(* CODESYS project tc3_bacnetrev14.library
   Company: Beckhoff Automation GmbH
   DefaultNamespace: Tc3_BACnetRev14
   Version: 4.0.18.1
   Placeholder: Tc3_BACnetRev14
   Author: Beckhoff Automation GmbH
   Description: The PLC library is a collection of function blocks for programming a BACnet controller. For each BACnet object function blocks are available that are read and written via the selected properties. In general a distinction is made between function blocks for server and client objects. Function blocks for client objects have the prefix "Remote", since they enable access to remote BACnet objects on other devices. The BACnet object function blocks ascertain whether process data are valid and the BACnet controller is ready for operation.
   Title: Tc3_BACnetRev14

Project tree, tasks and I/O mapping:
  libraries: Tc2_Standard, * (Beckhoff Automation GmbH); Tc2_System, * (Beckhoff Automation GmbH); Tc2_Utilities, * (Beckhoff Automation GmbH); Tc3_BA2_Common, * (Beckhoff Automation GmbH); Tc3_Module, * (Beckhoff Automation GmbH)
  DUTs/
    Enumerations/
      [Functional]/
        data type E_BACnet_CommMode
        data type E_BACnet_CreateObjType
        data type E_BACnet_EvaluationMode
        data type E_BACnet_ServerState
      [Internal]/
        data type E_BACnet_DeviceData
        data type E_BACnet_MultistateVal
        data type E_BACnet_PlcAction
      Properties/
        Error/
          data type E_BACnet_ErrorClass
          data type E_BACnet_ErrorCode
          data type E_BACnet_ErrorType
        Event/
          data type E_BACnet_EventState
          data type E_BACnet_EventTransitionBits
          data type E_BACnet_EventType
        Recipient/
          data type E_BACnet_AddressChoice
          data type E_BACnet_RecipientChoice
        Types/
          Calendar/
            data type E_BACnet_CalendarEntryChoice
            data type E_BACnet_CalendarEntryType
          DateTime/
            data type E_BACnet_DaysOfWeekBits
            data type E_BACnet_TimeStampChoice
          LogBuffer/
            data type E_BACnet_LogRecordChoice
          Scheduler/
            data type E_BACnet_EnumerationValueChoice
            data type E_BACnet_SchedBType
            data type E_BACnet_SpecialEventChoice
            data type E_BACnet_ValueChoice
          data type E_BACnet_BinaryPV
          data type T_BACnet_MultistateValue
        data type E_BACnet_AbortReason
        data type E_BACnet_AdapterStatus
        data type E_BACnet_ClientCOVChoice
        data type E_BACnet_DataTypes
        data type E_BACnet_DeviceStatus
        data type E_BACnet_FileAccessMethod
        data type E_BACnet_LifeSafetyMode
        data type E_BACnet_LifeSafetyOperation
        data type E_BACnet_LimitEnableBits
        data type E_BACnet_LoopMode
        data type E_BACnet_NodeType
        data type E_BACnet_NotifyType
        data type E_BACnet_ObjectSupportedBits
        data type E_BACnet_PersistentDataState
        data type E_BACnet_Priority
        data type E_BACnet_ProgramError
        data type E_BACnet_ProgramRequest
        data type E_BACnet_ProgramState
        data type E_BACnet_RejectReason
        data type E_BACnet_RestartReason
        data type E_BACnet_ScaleChoice
        data type E_BACnet_Segmentation
        data type E_BACnet_ServicesSupportedBits
        data type E_BACnet_SilencedState
        data type E_BACnet_StatusFlags
        data type E_BACnet_StringEncodingTypes
      Remote/
        data type E_BACnetRM_ClientState
        data type E_BACnetRM_RequestType
      data type E_BACnet_Error
    Interfaces/
      Remote/
        Objects/
          [Base]/
            interface I_BACnetRM_Object
          [Internal]/
            interface I_BACnetRM_BaseObject: OnCOV, OnReqError, Error, ObjectID, ObjectInstance, ObjectType, ReadMode
            interface I_BACnetRM_ObjectOwner: OnBACnetRMObjectCOV, OnBACnetRMObjectStateChanged, LogMsg
        Requests/
          [Base]/
            interface I_BACnetRM_BaseReq: Send, GetRequestType, IsReady
            interface I_BACnetRM_BasicReq: SetError, SetReady
      Server/
        [Base]/
          interface I_BACnet_Object: NextSibling, PrevSibling, IsDynamic, Parent, Description, ObjectName
        [Internal]/
          interface I_BACnet_BaseObject: NextObject, Error, ObjectID, ObjectInstance, ObjectType, Ready, ReadProperty, SyncPropertyCOV, WriteProperty
          interface I_BACnet_ObjectOwner: LogMsg, SymbolName, SymbolPath, OnBACnetObjectStateChanged
        Misc/
          interface I_BACnet_Cal
          interface I_BACnet_View: AddObject, RemoveObject, FindObject
    Types/
      [ADS]/
        data type ST_BACnet_AdsConnection
      [Functional]/
        data type U_BACnet_CreateObj
      Diagnose/
        data type ST_BACnet_ConfirmedServiceDiag
        data type ST_BACnet_DiagEthStatistics
        data type ST_BACnet_Diagnosis
        data type ST_BACnet_DiagnosisTiming
        data type ST_BACnet_FrameStatistics
        data type ST_BACnet_Info
        data type ST_BACnet_ServerStatistics
        data type ST_BACnet_TcIoEthStatistic
        data type ST_BACnet_TcIoEthTxRxErrorCount
        data type ST_BACnet_UnConfirmedServiceDiag
      Properties/
        [ADS]/
          Calendar/
            data type ST_BACnet_CalendarEntry
            data type ST_BACnet_CalendarEntryDate
            data type ST_BACnet_CalendarEntryDateRange
            data type ST_BACnet_CalendarEntryWeekNDay
            data type T_BACnet_CalendarEntryTypeFilter
          DateTime/
            data type ST_BACnet_TimeStampDateTime
            data type ST_BACnet_TimeValue
            data type ST_BACnet_TimeValueBool
            data type ST_BACnet_TimeValueList
            data type ST_BACnet_TimeValueReal
          LogBuffer/
            data type ST_BACnet_LogBufferEntryReal
            data type ST_BACnet_LogBufferReal
          LogRecord/
            data type ST_BACnet_LogDatum
            data type ST_BACnet_LogDatumList
            data type ST_BACnet_LogRecord
            data type ST_BACnet_LogRecordList
          Schedule/
            data type ST_BACnet_DailySchedule
            data type ST_BACnet_ExceptionScheduleBool
            data type ST_BACnet_ExceptionScheduleCalDate
            data type ST_BACnet_ExceptionScheduleCalRef
            data type ST_BACnet_ExceptionScheduleCalWnD
            data type ST_BACnet_ExceptionScheduleEntryBool
            data type ST_BACnet_ExceptionScheduleEntryReal
            data type ST_BACnet_ExceptionScheduleReal
            data type ST_BACnet_Value
            data type ST_BACnet_ValueList
          data type ST_BACnet_CharacterStringExt
          data type ST_BACnet_CharacterStringExtListEntry
          data type ST_BACnet_LimitEnable
          data type ST_BACnet_ObjectIdentifierList
        [Raw]/
          References/
            data type ST_BACnetRaw_DeviceObjectPropertyReference
            data type ST_BACnetRaw_DeviceObjectReference
            data type ST_BACnetRaw_ObjectPropertyReference
            data type ST_BACnetRaw_SetpointReference
          ValidFields/
            data type ST_BACnetRaw_ValidFields_DeviceObjectPropertyReference
        Accumulator/
          data type ST_BACnet_Prescale
          data type ST_BACnet_Scale
          data type ST_BACnet_ScaleValue
        Calendar/
          data type T_BACnet_CalendarDateList
        Event/
          data type ST_BACnet_Event
          data type ST_BACnet_EventMessageTexts
          data type ST_BACnet_EventMessageTextStrings
          data type ST_BACnet_Events
          data type ST_BACnet_EventTimeStamps
          data type T_BACnet_EventTransitions
          data type T_BACnet_EventTransitionTexts
        EventEnrollment/
          data type ST_BACnet_EventArguments
          data type ST_BACnet_EventBinaryCoded
          data type ST_BACnet_EventOutOfRange
          data type ST_BACnet_EventParameter
          data type ST_BACnet_EventUnsignedRange
        Recipient/
          data type ST_BACnet_Address
          data type ST_BACnet_Destination
          data type ST_BACnet_Recipient
          data type ST_BACnet_RecipientEntry
          data type ST_BACnet_ValidDays
          data type T_BACnet_RecipientList
        References/
          data type ST_BACnet_ObjectPropertyReference
        Scheduler/
          data type ST_BACnet_EnumerationValueType
          data type ST_BACnet_SchedCalendar
          data type ST_BACnet_SchedException
          data type ST_BACnet_SpecialEvent
          data type ST_BACnet_SpecialEventList
          data type T_BACnet_SchedCalendar
          data type T_BACnet_SchedExceptionEntryList
          data type T_BACnet_SchedExceptionList
          data type T_BACnet_SchedWeek
        TLog/
          data type T_BACnet_TLogBuffer
        data type ST_BACnet_ClientCOV
        data type ST_BACnet_EventTransitionBits
        data type ST_BACnet_LimitEnableBits
        data type ST_BACnet_ServicesSupportedBits
        data type ST_BACnet_StatusFlagBits
        data type T_BACnet_EventTransitionPriority
        data type T_BACnet_ObjectIdentifier
        data type T_BACnet_StateText
        data type T_BACnet_StateTextArray
      Remote/
        [Internal]/
          data type ST_BACnetRM_CmdRealValue
          data type ST_BACnetRM_FifoEntry
          data type ST_BACnetRM_LastWriteValue
          data type ST_BACnetRM_PropertyValueList
          data type ST_BACnetRM_ReadEntry
          data type ST_BACnetRM_ReqPtr
          data type ST_BACnetRM_RpmListEntry
          data type ST_BACnetRM_ScanParameter
          data type ST_BACnetRM_WriteEntry
        data type ST_BACnetRM_ScanResult
  GVLs/
    global variables BACnet_Globals
    global variables BACnet_Param
  POUs/
    Dynamic Objects/
      function block FB_BACnet_DynObjectManager [ST]: EvaluateStructure, DeleteObjectEx, OnPostOnlineChange, CreateObject, CreateObjectEx, DeleteObject, Ready, Reset, CreatedObjects, FB_exit
    Helper/
      [internal]/
        Calendar/
          function F_BACnet_ToDateListEntry [ST]
        Remote/
          function F_BACnetRM_GetWriteEntrySize [ST]
          function F_BACnetRM_IsErrorSet [ST]
          function F_IsCovProperty [ST]
          function F_IsCovReadMode [ST]
          function F_IsCovReqType [ST]
        Scheduler/
          function F_BA_CalendarSchedSize [ST]
          function F_BA_ExceptionSchedSize [ST]
        String/
          function F_BACnet_ChrStrExtLen [ST]
          function F_BACnet_DecodeUCS2 [ST]
          function F_BACnet_DecodeUCS4 [ST]
          function F_BACnet_DecodeUTF8 [ST]
          function F_BACnet_EncodeUTF8 [ST]
          function F_BACnet_GetUsedStateText [ST]
          function F_BACnet_GetUsedUDINT [ST]
          function F_BACnet_UCS2ToWin1252 [ST]
          function F_BACnet_Utf8ToWin1252 [ST]
          function F_BACnet_Win1252ToUCS2 [ST]
          function F_BACnet_Win1252ToUtf8 [ST]
        Validation-Functions/
          function F_BACnet_IsAbortReasonValid [ST]
          function F_BACnet_IsErrorClassValid [ST]
          function F_BACnet_IsErrorCodeValid [ST]
          function F_BACnet_IsErrorTypeValid [ST]
          function F_BACnet_IsObjIdentifierValid [ST]
          function F_BACnet_IsPriorityValid [ST]
          function F_BACnet_IsPropIdentifierValid [ST]
          function F_BACnet_IsRejectReasonValid [ST]
          function F_BACnet_IsSchedBTypeValid [ST]
        function F_BACnet_AlignedSize [ST]
        function F_BACnet_AnalogPV [ST]
        function F_BACnet_BitFieldBit [ST]
        function F_BACnet_ChangeBitFieldBit [ST]
        function F_BACnet_ElemSize [ST]
        function F_BACnet_EndOf [ST]
        function F_BACnet_FilterErrCode [ST]
        function F_BACnet_IsBitFieldBitSet [ST]
        function F_BACnet_IsBitFieldBitSetPtr [ST]
        function F_BACnet_NextListElem [ST]
        function F_BACnet_SetBitFieldBit [ST]
        function F_BACnet_SysTimeDiff [ST]
        function F_BACnet_UnSetBitFieldBit [ST]
      Flags/
        function F_BACnet_EventEnable [ST]
        function F_BACnet_EventTransitionFlags [ST]
        function F_BACnet_GetEventTransFlagsData [ST]
        function F_BACnet_GetLimitEnFlagsData [ST]
        function F_BACnet_GetStatusFlagsData [ST]
        function F_BACnet_LimitEnable [ST]
        function F_BACnet_LimitEnableFlags [ST]
        function F_BACnet_StatusFlags [ST]
      MultiState/
        function F_BACnet_EnMultiStatePV [ST]
        function F_BACnet_MultiStatePV [ST]
      NC/
        function F_BACnet_DeviceRecipient [ST]
        function F_BACnet_EthernetRecipient [ST]
        function F_BACnet_EthernetRecipientEx [ST]
      Real/
        function F_BACnet_EnRealPV [ST]
        function F_BACnet_IsFinite [ST]
        function F_BACnet_NAN [ST]
        function F_BACnet_RealEQ [ST]
        function F_BACnet_RealGE [ST]
        function F_BACnet_RealGT [ST]
        function F_BACnet_RealLE [ST]
        function F_BACnet_RealLT [ST]
        function F_BACnet_RealNothing [ST]
        function F_BACnet_RealNull [ST]
        function F_BACnet_RealPV [ST]
        function F_BACnet_RealToStr [ST]
      References/
        function F_BACnet_Reference [ST]
        function F_BACnet_ReferenceByID [ST]
      Schedule/
        Calendar/
          function F_BACnet_SchedCalendar [ST]
        Exception/
          function F_BACnet_SchedEntry1xA [ST]
          function F_BACnet_SchedEntry1xB [ST]
          function F_BACnet_SchedEntry1xM [ST]
          function F_BACnet_SchedEntry3xA [ST]
          function F_BACnet_SchedEntry3xB [ST]
          function F_BACnet_SchedEntry3xM [ST]
          function F_BACnet_SchedEntry5xA [ST]
          function F_BACnet_SchedEntry5xB [ST]
          function F_BACnet_SchedEntry5xM [ST]
        Weekly/
          function F_BACnet_SchedWeekly1xA [ST]
          function F_BACnet_SchedWeekly1xB [ST]
          function F_BACnet_SchedWeekly1xM [ST]
          function F_BACnet_SchedWeekly3xA [ST]
          function F_BACnet_SchedWeekly3xB [ST]
          function F_BACnet_SchedWeekly3xM [ST]
          function F_BACnet_SchedWeekly5xA [ST]
          function F_BACnet_SchedWeekly5xB [ST]
          function F_BACnet_SchedWeekly5xM [ST]
      String/
        function F_BACnet_GetObjectIdString [ST]
        function block FB_BACnet_StringExtDecode [ST]
        function block FB_BACnet_StringExtEncode [ST]
      function F_BACnet_GetObjectListIndex [ST]
      function F_BACnet_GetObjId [ST]
      function F_BACnet_GetObjInstance [ST]
      function F_BACnet_GetObjType [ST]
      function block FB_BACnet_AccLimit [ST]
      function block FB_BACnet_AvgValue [ST]
      function block FB_BACnet_PidControl [ST]
      function block FB_BACnet_PT1 [ST]
    Local/
      Objects/
        [Base]/
          Basic/
            function block FB_BACnet_EventObject [ST]: OnObjectStateChanged, OnPostInit, IsReliable, AcknowledgePLC, AcknowledgeRm, AckedTransitions, EventMessageTexts, EventState, EventTimeStamps, StatusFlags, FB_init
            function block FB_BACnet_Object [ST]: OnBACnetObjectStateChanged, OnCycle, RemoveFromLinkedObjList, LogMsg, NextSibling, PrevSibling, SymbolName, SymbolPath, Close, DynamicInit, OnObjectStateChanged, OnPostInit, ValidateReference, ConcatTitle, ValidateTitles, Parent, ReadPropertyExceptionSched, ReadPropertyReference, WritePropertyExceptionSched, WritePropertyReference, Description, ObjectName, FB_init
          function block FB_BACnet_BaseAcc [ST]: OnObjectStateChanged, FB_init
          function block FB_BACnet_BaseAI [ST]: OnObjectStateChanged, FB_init
          function block FB_BACnet_BaseAO [ST]: OnObjectStateChanged, ActivePrio, FB_init
          function block FB_BACnet_BaseBI [ST]: OnObjectStateChanged, ChangeOfStateTime, TimeOfActiveTimeReset, TimeOfStateCountReset, FB_init
          function block FB_BACnet_BaseBO [ST]: OnObjectStateChanged, ActivePrio, ChangeOfStateTime, TimeOfActiveTimeReset, TimeOfStateCountReset, FB_init
          function block FB_BACnet_BaseLoop [ST]: OnObjectStateChanged, ControlledVariable, ProportionalBand, Setpoint, FB_init
          function block FB_BACnet_BaseMI [ST]: OnObjectStateChanged, StateCount, FB_init
          function block FB_BACnet_BaseMO [ST]: OnObjectStateChanged, ActivePrio, StateCount, FB_init
          function block FB_BACnet_BasePC [ST]: OnObjectStateChanged, FB_init
          function block FB_BACnet_BaseSched [ST]: OnObjectStateChanged, ReadContent, WriteContent, ObjectPropertyReferences, FB_init
          function block FB_BACnet_BaseTLog [ST]: OnObjectStateChanged, LastNotifyRecord, RecordsSinceNotification
        [Internal]/
          5P/
            function block FB_BACnet_AO_5P [ST]: OnObjectStateChanged, EnManualOperator, ValManualOperator
            function block FB_BACnet_AO_IO5P [ST]: OnObjectStateChanged, EnManualOperator, ValManualOperator
            function block FB_BACnet_AO_Raw5P [ST]: OnObjectStateChanged, EnManualOperator, ValManualOperator
            function block FB_BACnet_AV_5P [ST]: OnObjectStateChanged, EnManualOperator, ValManualOperator
            function block FB_BACnet_BO_5P [ST]: OnObjectStateChanged, EnManualOperator, ValManualOperator
            function block FB_BACnet_BO_IO5P [ST]: OnObjectStateChanged, EnManualOperator, ValManualOperator
            function block FB_BACnet_BO_Raw5P [ST]: OnObjectStateChanged, EnManualOperator, ValManualOperator
            function block FB_BACnet_BV_5P [ST]: OnObjectStateChanged, EnManualOperator, ValManualOperator
            function block FB_BACnet_MO_5P [ST]: OnObjectStateChanged, EnManualOperator, ValManualOperator
            function block FB_BACnet_MO_IO5P [ST]: OnObjectStateChanged, EnManualOperator, ValManualOperator
            function block FB_BACnet_MO_Raw5P [ST]: OnObjectStateChanged, EnManualOperator, ValManualOperator
            function block FB_BACnet_MV_5P [ST]: OnObjectStateChanged, EnManualOperator, ValManualOperator
          Property/
            Buffer/
              [Archiv]/
                function block FB_BACnet_WeeklyScheduleBuffer [ST]: ResetValue, FB_init
              Base/
                function block FB_BACnet_BaseArrayBuffer [ST]
                function block FB_BACnet_BaseListBuffer [ST]: ValidateInst
                function block FB_BACnet_BasePropertyBuffer [ST]: MemSet, MemSetBYTE, MemSetUDINT, MemSetUINT, MemSetULINT, ReadValue, ValidateInst, WriteValue, OnObjectStateChanged, ResetValue
                function block FB_BACnet_BasePropertyLogBuffer [ST]: OnObjectStateChanged
              function block FB_BACnet_DateListBuffer [ST]: FB_init
              function block FB_BACnet_EventLogBuffer [ST]: ValidateInst, FB_init
              function block FB_BACnet_ExceptionScheduleBuffer [ST]: FB_init
              function block FB_BACnet_TLMBuffer [ST]: ValidateInst, ResetValue, FB_init
              function block FB_BACnet_TrendLogBuffer [ST]: ValidateInst, ResetValue, FB_init
          function block FB_BACnet_BaseObject [ST]: OnCycle, NextObject, View_AddSubordinate, View_RemoveSubordinate, Close, Sched_ReadEntry, Sched_SetNextDay, Sched_SetNextTimeVal, Sched_WriteEntry, DeleteObject, IsInitReady, OnObjectStateChanged, OnPostOnlineChange, Acknowledge, Error, IsDynamic, ObjectID, ObjectInstance, ObjectType, Ready, State, EnableProperty, SetPropertyCount, WriteProtectProperty, AddPropertyElement, AddPropertyElementPtr, RemoveArrayElements, RemoveListElements, SetNumberOfStates, ReadProperty, ReadPropertyAckedTransitions, ReadPropertyBool, ReadPropertyByte, ReadPropertyDateList, ReadPropertyEventEnable, ReadPropertyEventParameter, ReadPropertyEventState, ReadPropertyEventTimeStamps, ReadPropertyExceptionSched, ReadPropertyLimitEnable, ReadPropertyNotifyType, ReadPropertyReal, ReadPropertyRecipientList, ReadPropertyReference, ReadPropertyStatusFlags, ReadPropertyString, ReadPropertyUDInt, ReadPropertyUnit, ReadPropertyWeeklySched, AddListElement, ApplySyncHandler, EvaluatePropSync, IncrementSyncHandlers, RequestSyncHandlers, RequestSyncHandlersEx, SyncProperty, SyncPropertyCOV, SyncPropertyIdx, SyncPropertyList, SyncPropertyPvPrio, WriteProperty, WritePropertyBool, WritePropertyByte, WritePropertyDateList, WritePropertyEventEnable, WritePropertyEventParameter, WritePropertyExceptionSched, WritePropertyLimitEnable, WritePropertyNotifyType, WritePropertyNull, WritePropertyReal, WritePropertyRealPrio, WritePropertyRecipientList, WritePropertyReference, WritePropertyReferenceList, WritePropertyReferenceList1x, WritePropertyString, WritePropertyStringIdx, WritePropertyUDInt, WritePropertyUInt, WritePropertyUnit, WritePropertyValue, WritePropertyValueEx, WritePropertyWeeklySched, FB_exit
        Experimental/
          function block FB_BACnet_ExpEventLog [ST]
          function block FB_BACnet_ExpTLM [ST]: OnObjectStateChanged, FB_init
          function block FB_BACnet_ExpTLog [ST]: Trend_LastPlcTrendEntry, Trend_NextLogDatum, Trend_NextLogRecord, OnObjectStateChanged, ReadPropertyLogBuffer, WritePropertyLogBuffer, ObjectPropertyReference, FB_init
        Primitive/
          function block FB_BACnet_INT [ST]: OnObjectStateChanged, FB_init
          function block FB_BACnet_LAV [ST]: OnObjectStateChanged, FB_init
          function block FB_BACnet_String [ST]: OnObjectStateChanged, FB_init
          function block FB_BACnet_UINT [ST]: OnObjectStateChanged, FB_init
        function block FB_BACnet_Acc [ST]: OnObjectStateChanged, FB_init
        function block FB_BACnet_Acc_IO [ST]: OnObjectStateChanged, ValueBeforeChange, ValueChangeTime
        function block FB_BACnet_Acc_Raw [ST]: OnObjectStateChanged
        function block FB_BACnet_AI [ST]: OnObjectStateChanged
        function block FB_BACnet_AI_IO [ST]: OnObjectStateChanged
        function block FB_BACnet_AI_Raw [ST]: OnObjectStateChanged
        function block FB_BACnet_AO [ST]: OnObjectStateChanged
        function block FB_BACnet_AO_IO [ST]: OnObjectStateChanged
        function block FB_BACnet_AO_Raw [ST]: OnObjectStateChanged
        function block FB_BACnet_AV [ST]: OnObjectStateChanged, ActivePrio, FB_init
        function block FB_BACnet_AV_Disp [ST]: OnObjectStateChanged, FB_init
        function block FB_BACnet_AV_Setp [ST]: OnObjectStateChanged, FB_init
        function block FB_BACnet_BI [ST]: OnObjectStateChanged
        function block FB_BACnet_BI_IO [ST]: OnObjectStateChanged
        function block FB_BACnet_BI_Raw [ST]: OnObjectStateChanged
        function block FB_BACnet_BO [ST]: OnObjectStateChanged
        function block FB_BACnet_BO_IO [ST]: OnObjectStateChanged
        function block FB_BACnet_BO_Raw [ST]: OnObjectStateChanged
        function block FB_BACnet_BV [ST]: OnObjectStateChanged, ActivePrio, ChangeOfStateTime, TimeOfActiveTimeReset, TimeOfStateCountReset, FB_init
        function block FB_BACnet_BV_Disp [ST]: OnObjectStateChanged, FB_init
        function block FB_BACnet_BV_Setp [ST]: OnObjectStateChanged, FB_init
        function block FB_BACnet_Cal [ST]: OnObjectStateChanged, ReadContent, WriteContent, FB_init
        function block FB_BACnet_Device [ST]: OnObjectStateChanged, Location, FB_init
        function block FB_BACnet_EE [ST]: OnObjectStateChanged, ReadContent, WriteContent, ObjectPropertyReference, FB_init
        function block FB_BACnet_ELog [ST]: OnObjectStateChanged, FB_init
        function block FB_BACnet_File [ST]: OnObjectStateChanged, FB_init
        function block FB_BACnet_Loop [ST]: OnObjectStateChanged, ControlledVariable, Setpoint
        function block FB_BACnet_Loop_Ref [ST]: OnObjectStateChanged, ControlledVariable, ControlledVariableReference, ManipulatedVariableReference, Setpoint, SetpointReference
        function block FB_BACnet_MI [ST]: OnObjectStateChanged
        function block FB_BACnet_MI_IO [ST]: OnObjectStateChanged
        function block FB_BACnet_MI_Raw [ST]: OnObjectStateChanged
        function block FB_BACnet_MO [ST]: OnObjectStateChanged
        function block FB_BACnet_MO_IO [ST]: OnObjectStateChanged
        function block FB_BACnet_MO_Raw [ST]: OnObjectStateChanged
        function block FB_BACnet_MV [ST]: OnObjectStateChanged, ActivePrio, StateCount, FB_init
        function block FB_BACnet_MV_Disp [ST]: OnObjectStateChanged, StateCount, FB_init
        function block FB_BACnet_MV_Setp [ST]: OnObjectStateChanged, StateCount, FB_init
        function block FB_BACnet_NC [ST]: OnObjectStateChanged, FB_init
        function block FB_BACnet_PC [ST]: OnObjectStateChanged, InputReference, FB_init
        function block FB_BACnet_PC_Raw [ST]: OnObjectStateChanged, FB_init
        function block FB_BACnet_Prog [ST]: OnObjectStateChanged, FB_init
        function block FB_BACnet_SchedA [ST]: OnObjectStateChanged, FB_init
        function block FB_BACnet_SchedB [ST]: OnObjectStateChanged, FB_init
        function block FB_BACnet_SchedM [ST]: OnObjectStateChanged, FB_init
        function block FB_BACnet_TLM [ST]: OnObjectStateChanged, ObjectPropertyReferences, FB_init
        function block FB_BACnet_TLog [ST]: OnObjectStateChanged, ObjectPropertyReference, FB_init
        function block FB_BACnet_View [ST]: AddObject, RemoveObject, Close, OnObjectStateChanged, FindObject, FB_init
      function block FB_BACnet_Server [ST]: GetObjectByID, RegisterObject, ObjectCount, ServerItf, Reset, OnPostOnlineChange, Error, Operational, Valid, ReadPropertyInt, ReadPropertyUDInt, FB_Exit
    Remote/
      Objects/
        Basic/
          [Base]/
            Basic/
              function block FB_BACnetRM_Object [ST]: OnBACnetRMObjectCOV, OnBACnetRMObjectStateChanged, LogMsg, FB_init
            function block FB_BACnetRM_BaseTLog [ST]: OnObjectStateChanged
            function block FB_BACnetRM_EventObject [ST]: OnObjectStateChanged, StatusFlags
          [Internal]/
            function block FB_BACnetRM_BaseObject [ST]: OnCOV, OnReqError, OnObjectStateChanged, Error, ObjectID, ObjectInstance, ObjectType, ReadMode, SyncProperty, SyncPropertyEnable, SyncPropertyIdx, SyncPropertyPrio, SyncPropertyPrioReal, SyncPropertyReal
          function block FB_BACnetRM_Acc [ST]: OnObjectStateChanged, FB_init
          function block FB_BACnetRM_AI [ST]: OnObjectStateChanged, FB_init
          function block FB_BACnetRM_AO [ST]: OnObjectStateChanged, FB_init
          function block FB_BACnetRM_AV [ST]: OnObjectStateChanged, FB_init
          function block FB_BACnetRM_AV_Disp [ST]: OnObjectStateChanged, FB_init
          function block FB_BACnetRM_AV_Setp [ST]: OnCOV, OnObjectStateChanged, FB_init
          function block FB_BACnetRM_Avg [ST]: OnObjectStateChanged, FB_init
          function block FB_BACnetRM_BI [ST]: OnObjectStateChanged, FB_init
          function block FB_BACnetRM_BO [ST]: OnObjectStateChanged, FB_init
          function block FB_BACnetRM_BV [ST]: OnObjectStateChanged, FB_init
          function block FB_BACnetRM_BV_Disp [ST]: OnObjectStateChanged, FB_init
          function block FB_BACnetRM_BV_Setp [ST]: OnCOV, OnObjectStateChanged, FB_init
          function block FB_BACnetRM_Cal [ST]: OnObjectStateChanged, FB_init
          function block FB_BACnetRM_Cmd [ST]: OnObjectStateChanged, FB_init
          function block FB_BACnetRM_Device [ST]: OnObjectStateChanged, FB_init
          function block FB_BACnetRM_EE [ST]: OnObjectStateChanged, FB_init
          function block FB_BACnetRM_ELog [ST]: FB_init
          function block FB_BACnetRM_File [ST]: OnObjectStateChanged, FB_init
          function block FB_BACnetRM_Group [ST]: OnObjectStateChanged, FB_init
          function block FB_BACnetRM_Loop [ST]: OnObjectStateChanged, FB_init
          function block FB_BACnetRM_MI [ST]: OnObjectStateChanged, FB_init
          function block FB_BACnetRM_MO [ST]: OnObjectStateChanged, FB_init
          function block FB_BACnetRM_MV [ST]: OnObjectStateChanged, FB_init
          function block FB_BACnetRM_MV_Disp [ST]: OnObjectStateChanged, FB_init
          function block FB_BACnetRM_MV_Setp [ST]: OnCOV, OnObjectStateChanged, FB_init
          function block FB_BACnetRM_NC [ST]: FB_init
          function block FB_BACnetRM_PC [ST]: OnObjectStateChanged, FB_init
          function block FB_BACnetRM_Prog [ST]: OnObjectStateChanged, FB_init
          function block FB_BACnetRM_SchedA [ST]: OnObjectStateChanged, FB_init
          function block FB_BACnetRM_SchedB [ST]: OnObjectStateChanged, FB_init
          function block FB_BACnetRM_SchedM [ST]: OnObjectStateChanged, FB_init
          function block FB_BACnetRM_TLM [ST]: OnObjectStateChanged, FB_init
          function block FB_BACnetRM_TLog [ST]: OnObjectStateChanged, FB_init
        Convenience/
          function block FB_BACnetRM_CnvLoop [ST]: OnObjectStateChanged
        Experimental/
          function block FB_BACnetRM_ExpAV01 [ST]: OnObjectStateChanged
          function block FB_BACnetRM_ExpAV02 [ST]
        Primitive/
          function block FB_BACnetRM_BitString [ST]: OnObjectStateChanged, FB_init
          function block FB_BACnetRM_ByteArr [ST]: OnObjectStateChanged, FB_init
          function block FB_BACnetRM_Date [ST]: OnObjectStateChanged, FB_init
          function block FB_BACnetRM_DateP [ST]: OnObjectStateChanged, FB_init
          function block FB_BACnetRM_DateTime [ST]: OnObjectStateChanged, FB_init
          function block FB_BACnetRM_DateTimeP [ST]: OnObjectStateChanged, FB_init
          function block FB_BACnetRM_Int [ST]: OnObjectStateChanged, FB_init
          function block FB_BACnetRM_LAV [ST]: OnObjectStateChanged, FB_init
          function block FB_BACnetRM_String [ST]: OnObjectStateChanged, FB_init
          function block FB_BACnetRM_Time [ST]: OnObjectStateChanged, FB_init
          function block FB_BACnetRM_TimeP [ST]: OnObjectStateChanged, FB_init
          function block FB_BACnetRM_UInt [ST]: OnObjectStateChanged, FB_init
      Properties/
        [Base]/
          function block FB_BACnetRM_BaseProperty [ST]: SetBusy, SetError, SetReady, OnExecuteChange, Free, Busy, Error, Ready, Request, Valid
        function block FB_BACnetRM_ReadProperty [ST]: OnExecuteChange, Free, Valid, FB_exit
        function block FB_BACnetRM_ReadPropertyEx [ST]
        function block FB_BACnetRM_WriteProperty [ST]: OnExecuteChange, Free, Valid, FB_exit
        function block FB_BACnetRM_WritePropertyEx [ST]
      Requests/
        [Internal]/
          [Base]/
            function block FB_BACnetRM_ReqBase [ST]: OnError, Valid, GetRequestType, IsReady, Send
            function block FB_BACnetRM_ReqBasic [ST]: OnSendPropertyDataRequest, InitTimer, SetBusy, SetError, SetReady, TcAddRef, TcQueryInterface, TcRelease, CopyRemoteData, ProcessResult, Send, StartTimer, GetRequestType, IsReady
          function block FB_BACnetRM_ReqAckAlarm [ST]: OnSendPropertyDataRequest, Send, TcAddRef, TcQueryInterface, TcRelease, UpdateTimeStamp, GetRequestType, IsReady
          function block FB_BACnetRM_ReqCov [ST]: AddCovSlave, Send, ProcessResult, StartTimer, GetRequestType, IsReady, FB_Exit, Master, SendSubscription
          function block FB_BACnetRM_ReqFifo [ST]: AddFifoReq, ProcessReadFifo, ProcessWriteFifo, Valid, FB_Exit
          function block FB_BACnetRM_ReqListAdd [ST]: Send, ProcessResult, GetRequestType, IsReady
          function block FB_BACnetRM_ReqListRem [ST]: Send, ProcessResult, GetRequestType
          function block FB_BACnetRM_ReqRead [ST]: Send, OnError, ProcessResult, GetRequestType
          function block FB_BACnetRM_ReqRpm [ST]: Send, UpdateRequest, Free, OnError, ProcessResult, GetRequestType, _WritePropEntry, FB_exit
          function block FB_BACnetRM_ReqWpm [ST]: Send, UpdateRequest, Free, OnError, ProcessResult, GetRequestType, FB_exit
          function block FB_BACnetRM_ReqWrite [ST]: Send, OnError, ProcessResult, GetRequestType, IsReady
      function block FB_BACnet_Client [ST]: OnCOV, OnReqError, OnRequestComplete, AddReadEntry, AddWriteEntry, AddFifoReadReq, AddFifoWriteReq, UpdateRequests, CreateReadReq, CreateReqList, DeleteReqList, OptimizeCOV, OnPostOnlineChange, Error, ObjectID, ObjectInstance, ObjectType, OpenRequestCount, ReadMode, Ready, State, FB_Exit
    function block FB_BACnet_Adapter [ST]: GetDiagnosis, ResetDiagnosis, Device, Error, GetScanResult, StartScan, StartScanEx, TimeSync, FB_exit, FB_init
  TEST/
    TestPackage/
      Samples/
        Objects/
          Local/
            function block FB_BACnet_SmplAV01 [ST]: OnObjectStateChanged
            function block FB_BACnet_SmplBO01 [ST]
          Remote/
            function block FB_BACnetRM_SmplAV01 [ST]: OnObjectStateChanged
        Project Structure/
          PRG02/
            TEMPLATES/
              Custom/
                H/
                  HtgCirABC123/
                    function block FB_BA_HtgCirABC123 [CFC]: FB_init
                    function block FB_BA_HtgCirABC123_Vlv [CFC]: FB_init
                  HtgCirTZU555/
                    function block FB_BA_HtgCirTZU555 [CFC]: FB_init
                    function block FB_BA_HtgCirTZU555_Pu [CFC]: FB_init
              Standard/
                AC/
                  function block FB_BACnet_AC01 [CFC]: FB_init
                H/
                  function block FB_BACnet_HtgCir01 [CFC]: FB_init
                Universal/
                  Valve/
                    function block FB_Bnet_Vlv_014 [CFC]: FB_init
            program MAIN_PRG02 [ST]
      Templates/
        HeatSupply/
          HeatingCircuit/
            Plants/
              function block FB_Bnet_H_HtgCir_01 [CFC]: FB_init
            function block FB_Bnet_H_HtgCir_HtgLmt [CFC]: FB_init
            function block FB_Bnet_H_HtgCir_Sp [CFC]: FB_init
            function block FB_MMUX_R04 [ST]
            function block FB_Swi2P [ST]
          data type E_xEnergyLvl
          data type E_xEnergyLvlA
          function block FB_Bnet_H_OpM [CFC]: FB_init
          function block FB_PrioSwi_B04 [ST]
          function block FB_PrioSwi_UDI08 [ST]
        Internal/
          function block FB_BACnet_Server_NC01 [ST]
        Universal/
          AntiBlocking/
            function F_RemSecsTon [ST]
            function block FB_AntBlkg [ST]
            function block FB_Bnet_AntiBlocking [CFC]: FB_init
          Control/
            DelayOff/
              function block FB_Bnet_DlyOff [CFC]: FB_init
            Scale/
              function block FB_Bnet_Scale_04 [CFC]: FB_init
              function block FB_Chrct04 [ST]
          Pump/
            1st/
              function block FB_Bnet_Pu1st [CFC]: FB_init
          Valve/
            function block FB_Bnet_Vlv_013 [CFC]: FB_init
        global variables Const
      TestFBs/
        RT/
          function block FB_ArrayHtgCir [ST]: FB_init
          function block FB_ArrayTest [ST]: FB_init
        function block FB_ClientTest [ST]
      program _MAIN [ST]
      program BACKUP [ST]
      program CLIENT [ST]
      program DYN_OBJECTS [ST]
      program PERFORMANCE [ST]
      program PERFORMANCE_MIX [ST]
      program PLANT_DEMO [ST]: FB_init
      program RT [ST]
    program CLIENT_Andreas [ST]
    program CLIENT_Marco [ST]
    program Experimental [ST]
    program MAIN [ST]
    program TEMP [ST]
  Version/
    global variables Global_Version
*)

// DUTs/Enumerations/[Functional]/E_BACnet_CommMode
{attribute 'qualified_only'}
TYPE E_BACnet_CommMode :
(
	eAuto	:= 0,
	
	eCov	:= 1,
	eCovC	:= 2,
	eCovU	:= 3,
	eRp		:= 4,
	eRpm	:= 5
);
END_TYPE

// DUTs/Enumerations/[Functional]/E_BACnet_CreateObjType
{attribute 'qualified_only'}
TYPE E_BACnet_CreateObjType:
(
	eAnalogInputRaw,
	eAnalogOutputRaw,
	eAnalogOutputRaw5P,
	eAnalogValue,
	eAnalogValue5P,
	eAnalogValueDisp,
	eAnalogValueSetp,
	
	eBinaryInputRaw,
	eBinaryOutputRaw,
	eBinaryOutputRaw5P,
	eBinaryValue,
	eBinaryValue5P,
	eBinaryValueDisp,
	eBinaryValueSetp,
	
	eMultiStateInputRaw,
	eMultiStateOutputRaw,
	eMultiStateOutputRaw5P,
	eMultiStateValue,
	eMultiStateValue5P,
	eMultiStateValueDisp,
	eMultiStateValueSetp,
	
	eCalendar,
	eDevice,
	eFile,
	eLoop,
	eNotificationClass,
	eProg,
	eScheduleAnalog,
	eScheduleBinary,
	eScheduleMultistate,
	eAccumulator,
	ePulseConverter,
	eStructuredView
);
END_TYPE

// DUTs/Enumerations/[Functional]/E_BACnet_EvaluationMode
{attribute 'hide'}
{attribute 'qualified_only'}
TYPE E_BACnet_EvaluationMode :
(
	// [Management] Dynamic Objects:
	eDeleteObjects			:= 0,
	eCycle					:= 1
);
END_TYPE

// DUTs/Enumerations/[Functional]/E_BACnet_ServerState
{attribute 'qualified_only'}
TYPE E_BACnet_ServerState :
(
	Invalid					:= 0,
	
	eInitServer				:= 1,
	eInitDefObjs			:= 2,
	eInitUndefObjs			:= 3,
	eInitDefRefObjs			:= 4,
	eInitUndefRefObjs		:= 5,
	eOperation				:= 6
	
) BYTE;
END_TYPE

// DUTs/Enumerations/[Internal]/E_BACnet_DeviceData
{attribute 'hide'}
{attribute 'qualified_only'}
TYPE E_BACnet_DeviceData :
(
	eGetDiagnosis	:= 16#00000001,
	eResetDiagnosis	:= 16#80000001,
	eGetScanResult	:= 16#00000002,
	eGetIPSettings	:= 16#00000003,
	eSetIPSettings	:= 16#80000003,
	eGetBDT			:= 16#00000004,
	eSetBDT			:= 16#80000004,
	eGetFDT			:= 16#00000005,
	eSetPlcOID		:= 16#80000006,
	eSetPlcAdsPort	:= 16#80000007
	
) UDINT;
END_TYPE

// DUTs/Enumerations/[Internal]/E_BACnet_MultistateVal
{attribute 'hide'}
{attribute 'qualified_only'}
TYPE E_BACnet_MultistateVal:
(
	eNull					:= 16#0,
	eMin					:= 1,
	eNothing				:= 16#FFFFFFFF
) UDINT;
END_TYPE

// DUTs/Enumerations/[Internal]/E_BACnet_PlcAction
{attribute 'hide'}
{attribute 'qualified_only'}
TYPE E_BACnet_PlcAction :
(
	eIdle,
	eStart,
	eSuspend,
	eCreateFinish
) UINT;
END_TYPE

// DUTs/Enumerations/Properties/Error/E_BACnet_ErrorClass
{attribute 'qualified_only'}
{warning disable C0125}
TYPE E_BACnet_ErrorClass :
(
	eDevice					:= 0,
	eObject					:= 1,
	eProperty				:= 2,
	eResources				:= 3,
	eSecurity				:= 4,
	eServices				:= 5,
	eVt						:= 6,
	eCommunication			:= 7,
	
	eErrorClassUnknown	    := 255,
	
	NoError					:= 256,
	First					:= eDevice,
	Last					:= eCommunication,
	Count					:= (Last - First + 1)
);
END_TYPE
{warning restore C0125}

// DUTs/Enumerations/Properties/Error/E_BACnet_ErrorCode
{attribute 'qualifiedOnly'}
{warning disable C0125}
TYPE E_BACnet_ErrorCode :
(
	eOther										:= 0,
	eAuthenticationFailed						:= 1,
	eConfigurationInProgress					:= 2,
	eDeviceBusy									:= 3,
	eDynamicCreationNotSupported				:= 4,
	eFileAccessDenied							:= 5,
	eIncompatibleSecurityLevels					:= 6,
	eInconsistentParameters						:= 7,
	eInconsistentSelectionCriterion				:= 8,
	eInvalidDataType							:= 9,
	eInvalidFileAccessMethod					:= 10,
	eInvalidFileStartPosition					:= 11,
	eInvalidOperatorName						:= 12,
	eInvalidParameterDataType					:= 13,
	eInvalidTimeStamp							:= 14,
	eKeyGenerationError							:= 15,
	eMissingRequiredParameter					:= 16,
	eNoObjectsOfSpecifiedType					:= 17,
	eNoSpaceForObject							:= 18,
	eNoSpaceToAddListElement					:= 19,
	eNoSpaceToWriteProperty						:= 20,
	eNoVTSessionsAvailable						:= 21,
	ePropertyIsNotAList							:= 22,
	eObjectDeletionNotPermitted					:= 23,
	eObjectIdentifierAlreadyExists				:= 24,
	eOperationalProblem							:= 25,
	ePasswordFailure							:= 26,
	eReadAccessDenied							:= 27,
	eSecurityNotSupported						:= 28,
	eServiceRequestDenied						:= 29,
	eTimeout									:= 30,
	eUnknownObject								:= 31,
	eUnknownProperty							:= 32,
	eUnknownVTClass								:= 34,
	eUnknownVTSession							:= 35,
	eUnsupportedObjectType						:= 36,
	eValueOutOfRange							:= 37,
	eVtSessionAlreadyClosed						:= 38,
	eVtSessionTerminationFailure				:= 39,
	eWriteAccessDenied							:= 40,
	eCharacterSetNotSupported					:= 41,
	eInvalidArrayIndex							:= 42,
	eCovSubscriptionFailed						:= 43,
	eNotCovProperty								:= 44,
	eOptionalFunctionalityNotSupported			:= 45,
	eInvalidConfigurationData					:= 46,
	eDatatypeNotSupported						:= 47,
	eDuplicateName								:= 48,
	eDuplicateObjectId							:= 49,
	ePropertyIsNotAnArray						:= 50,
	eAbortBufferOverflow						:= 51,
	eAbortInvalidAPDUInThisState				:= 52,
	eAbortPreemptedByHigherPriorityTask			:= 53,
	eAbortSegmentationNotSupported				:= 54,
	eAbortProprietary							:= 55,
	eAbortOther									:= 56,
	eInvalidTag									:= 57,
	eNetworkDown								:= 58,
	eRejectBufferOverflow						:= 59,
	eRejectInconsistentParameters				:= 60,
	eRejectInvalidParameterDataType				:= 61,
	eRejectInvalidTag							:= 62,
	eRejectMissingRequiredParameter				:= 63,
	eRejectParameterOutOfRange					:= 64,
	eRejectTooManyArguments						:= 65,
	eRejectUndefinedEnumeration					:= 66,
	eRejectUnrecognizedService					:= 67,
	eRejectProprietary							:= 68,
	eRejectOther								:= 69,
	eUnknownDevice								:= 70,
	eUnknownRoute								:= 71,
	eValueNotInitialized						:= 72,
	eInvalidEventState							:= 73,
	eNoAlarmConfigured							:= 74,
	eLogBufferFull								:= 75,
	eLoggedValuePurged							:= 76,
	eNoPropertySpecified						:= 77,
	eNotConfiguredForTriggeredLogging			:= 78,
	eUnknownSubscription						:= 79,
	eParameterOutOfRange						:= 80,
	eListElementNotFound						:= 81,
	eBusy										:= 82,
	eCommunicationDisabled						:= 83,
	eUnknownFileSize							:= 122,
	eAbortAPDUTooLong							:= 123,
	eAbortApplicationExceededReplyTime			:= 124,
	eAbortOutOfResources						:= 125,
	eAbortTsmTimeout							:= 126,
	eAbortWindowSizeOutOfRange					:= 127,
	eFileFull									:= 128,
	eInconsistentConfiguration					:= 129,
	eInconsistentObjectType						:= 130,
	eInternalError								:= 131,
	eNotConfigured								:= 132,
	eOutOfMemory 								:= 133,
	
	NoError										:= 256,
	First										:= eOther,
	Last										:= eOutOfMemory,
	Count										:= (Last - First + 1)
);
END_TYPE
{warning restore C0125}

// DUTs/Enumerations/Properties/Error/E_BACnet_ErrorType
{attribute 'qualified_only'}
{warning disable C0125}
TYPE E_BACnet_ErrorType :
(
	eError,
	eReject,
	eAbort,
	
	First					:= eError,
	Last					:= eAbort,
	Count					:= (Last - First + 1)
);
END_TYPE
{warning restore C0125}

// DUTs/Enumerations/Properties/Event/E_BACnet_EventState
{attribute 'qualified_only'}
TYPE E_BACnet_EventState:
(
	eNormal := 0,
	eFault := 1,
	eOffnormal := 2,
	eHighLimit := 3,
	eLowLimit := 4,
	eLifeSafetyAlarm := 5
) UDINT;
END_TYPE

// DUTs/Enumerations/Properties/Event/E_BACnet_EventTransitionBits
{attribute 'qualified_only'}
TYPE E_BACnet_EventTransitionBits:
(
	Invalid			:= -1,
	
	eToOffnormal	:= 0,
	eToFault		:= 1,
	eToNormal		:= 2
);
END_TYPE

// DUTs/Enumerations/Properties/Event/E_BACnet_EventType
{attribute 'qualified_only'}
TYPE E_BACnet_EventType:
(
	Invalid := -1,
	
	eChangeOfBitstring := 0,
	eChangeOfState := 1,
	eChangeOfValue := 2,
	eCommandFailure := 3,
	eFloatingLimit := 4,
	eOutOfRange := 5,
	eComplexEventType := 6,
	eDeprecated7 := 7,
	eChangeOfLifeSafety := 8,
	eEnumeration := 9,
	eBufferReady := 10,
	eUnsignedRange := 11,
	eReserved12 := 12,
	eAccessEvent := 13,
	eDoubleOutOfRange := 14,
	eSignedOutOfRange := 15,
	eUnsignedOutOfRange := 16,
	eChangeOfCharacterstring := 17,
	eChangeOfStateFlags := 18,
	eChangeOfReliability := 19
);
END_TYPE

// DUTs/Enumerations/Properties/Recipient/E_BACnet_AddressChoice
{attribute 'qualified_only'}
TYPE E_BACnet_AddressChoice :
(
	eEthernet:=0,
	eArcnet:=1,
	eMsTp:=2,
	eLonTalk:=3,
	eLonTalkNeuronId:=4,
	eAddress_3:=5,
	eAddress_4:=6,
	eAddress_5:=7,
	eBroadcast:=8
);
END_TYPE

// DUTs/Enumerations/Properties/Recipient/E_BACnet_RecipientChoice
{attribute 'qualified_only'}
TYPE E_BACnet_RecipientChoice :
(
	eDevice,
	eAddress
);
END_TYPE

// DUTs/Enumerations/Properties/Types/Calendar/E_BACnet_CalendarEntryChoice
{attribute 'qualified_only'}
TYPE E_BACnet_CalendarEntryChoice :
(
(*
	BACnetDate              DATE;
	BACnetDateRange   		dateRange;
	BACnetWeekNDay          weekNDay;
*)
	eDate,
	eDateRange,
	eWeekNDay
);
END_TYPE

// DUTs/Enumerations/Properties/Types/Calendar/E_BACnet_CalendarEntryType
{attribute 'qualified_only'}
TYPE E_BACnet_CalendarEntryType : (* Not a BACnet-Stack type! *)
(
	eNone,
	eRef,
	eDate,
	eDateRange,
	eWeekNDay
);
END_TYPE

// DUTs/Enumerations/Properties/Types/DateTime/E_BACnet_DaysOfWeekBits
{attribute 'qualified_only'}
TYPE E_BACnet_DaysOfWeekBits :
(
	Invalid		:= -1,
	
	eBitMonday		:= 0,
	eBitTuesday		:= 1,
	eBitWednesday	:= 2,
	eBitThursday	:= 3,
	eBitFriday		:= 4,
	eBitSaturday	:= 5,
	eBitSunday		:= 6
);
END_TYPE

// DUTs/Enumerations/Properties/Types/DateTime/E_BACnet_TimeStampChoice
{attribute 'qualified_only'}
TYPE E_BACnet_TimeStampChoice :
(
	eTsTime,
    eSequenceNumber,
    eDateTime
);
END_TYPE

// DUTs/Enumerations/Properties/Types/LogBuffer/E_BACnet_LogRecordChoice
{attribute 'qualified_only'}
TYPE E_BACnet_LogRecordChoice :
(
(*
enum BACnetLogRecordChoice
{
      logStatus,              // [0] BACnetLogStatus,
      booleanValue,           // [1] BOOL,
      realValue,              // [2] REAL,
      enumValue,              // [3] ENUMERATED, __ Optionally limited to 32 bits
      unsignedValue,          // [4] Unsigned, __ Optionally limited to 32 bits
      signedValue,            // [5] INTEGER, __ Optionally limited to 32 bits
      bitstringValue,         // [6] BIT STRING, __ Optionally limited to 32 bits
      nullValue,              // [7] NULL,
      failure,                // [8] Error,
      timeChange,             // [9] REAL,
      anyValue,               // [10] ABSTRACT_SYNTAX.&Type __ Optional
};
*)
	eLogStatus 	:= 0, (* BACnetLogStatus *)
	eBooleanValue := 1, (*  BOOL, *)
	eRealValue	:= 2, (*  REAL, *)
	eEnumValue	:= 3, (*  ENUMERATED, __ Optionally limited TO 32 bits *)
	eUnsignedValue:= 4, (*  Unsigned, __ Optionally limited TO 32 bits *)
	eSignedValue	:= 5, (*  INTEGER, __ Optionally limited TO 32 bits *)
	eBitstringValue:= 6, (*  BIT STRING, __ Optionally limited TO 32 bits *)
	eNullValue	:= 7, (*  NULL, *)
	eFailure		:= 8, (*  Error, *)
	eTimeChange	:= 9, (*  REAL, *)
	eAnyValue		:= 10 (*  ABSTRACT_SYNTAX.&TYPE __ Optional *)
);
END_TYPE

// DUTs/Enumerations/Properties/Types/Scheduler/E_BACnet_EnumerationValueChoice
{attribute 'qualified_only'}
TYPE E_BACnet_EnumerationValueChoice :
(
	  eEnum := 0,
      eBinaryPV := 1,
      eEngineeringUnits := 2
)UDINT;
END_TYPE

// DUTs/Enumerations/Properties/Types/Scheduler/E_BACnet_SchedBType
{attribute 'qualified_only'}
{warning disable C0125}
TYPE E_BACnet_SchedBType :
(
	Invalid				:= 0,
	
	eBinaryPV			:= 1,
	eBool				:= 2,
	
	First				:= eBinaryPV,
	Last				:= eBool,
	Count				:= (Last - First + 1)
);
END_TYPE
{warning restore C0125}

// DUTs/Enumerations/Properties/Types/Scheduler/E_BACnet_SpecialEventChoice
{attribute 'qualified_only'}
TYPE E_BACnet_SpecialEventChoice :
(
	eCalendarEntry,
	eCalendarReference
);
END_TYPE

// DUTs/Enumerations/Properties/Types/Scheduler/E_BACnet_ValueChoice
{attribute 'qualified_only'}
{warning disable C0125}
TYPE E_BACnet_ValueChoice :
(
	Invalid						:= -1,
	
	eNullValue					:= 0,
	eBoolValue					:= 1,
	eUnsignedValue				:= 2,
	eSignedValue				:= 3,
	eRealValue					:= 4,
	eDoubleValue				:= 5,
	eOctedStringValue			:= 6,
	eCharStringValue			:= 7,
	eObjectIdentifierValue 		:= 8,		// but DataType is 0x0C
	eEnumerationValue			:= 9,
	eMaxBACnetValueChoice		:= 10
	
	//XFirst						:= eNullValue,
	//XLast						:= eMaxBACnetValueChoice,
	//Count						:= (Last - First + 1)
);
END_TYPE
{warning restore C0125}

// DUTs/Enumerations/Properties/Types/E_BACnet_BinaryPV
{attribute 'qualified_only'}
TYPE E_BACnet_BinaryPV:
(
	eInactive := 0,
	eActive := 1,
	eNull := 2,
	eNothing := 16#FFFF
);
END_TYPE

// DUTs/Enumerations/Properties/Types/T_BACnet_MultistateValue
TYPE T_BACnet_MultistateValue : ARRAY[1..BACnet_Param.nMultistate_StateCount] OF UDINT; END_TYPE

// DUTs/Enumerations/Properties/E_BACnet_AbortReason
{attribute 'qualified_only'}
{warning disable C0125}
TYPE E_BACnet_AbortReason :
(
	Invalid								:= -1,
	NoReason							:= 256,
	
	eOther								:= 0,
	eBufferOverflow						:= 1,
	eInvalidAPDUInThisState				:= 2,
	ePreemptedByHigherPriorityTask		:= 3,
	eSegmentationNotSupported			:= 4,
	eWindowSizeOutOfRange				:= 7,
	eApplicationExceededReplyTime		:= 8,
	eOutOfResources						:= 9,
	eTSMTimeout							:= 10,
	eAPDUTooLong						:= 11,
	
	First								:= eOther,
	Last								:= eAPDUTooLong,
	Count								:= (Last - First + 1)
);
END_TYPE
{warning restore C0125}

// DUTs/Enumerations/Properties/E_BACnet_AdapterStatus
{attribute 'qualified_only'}
TYPE E_BACnet_AdapterStatus :
(
	eInit				:= 16#0,
	eCheckIpAddr		:= 16#1,
	eCheckParam			:= 16#2,
	eGetGatewayMAC		:= 16#3,
	eWaitGatewayMAC		:= 16#4,
	eComplete			:= 16#8
);
END_TYPE

// DUTs/Enumerations/Properties/E_BACnet_ClientCOVChoice
{attribute 'qualified_only'}
{attribute 'strict'}
TYPE E_BACnet_ClientCOVChoice :
(
	eCovNull := 0,
	eCovReal := 1
);
END_TYPE

// DUTs/Enumerations/Properties/E_BACnet_DataTypes
{attribute 'qualified_only'}
TYPE E_BACnet_DataTypes:
(
	Invalid := -1,
	
	eNull := 0,
	eBool := 1,
	eUnsignedInteger := 2,
	eSignedInteger := 3,
	eReal := 4,
	eDouble := 5,
	eOctetString := 6,
	eCharacterStringExt := 7,
	eBitString := 8,
	eEnumerated := 9,
	eDate := 10,
	eTime := 11,
	eObjectIdentifier := 12,
	eDateTime := 14,
	eArrayIndex := 15,
	eCalendarEntry := 16,
	eObjectType := 17,
	eEventTransitionBits := 18,
	eActionList := 19,
	eStatusFlags := 20,
	eEventState := 21,
	eReliability := 22,
	ePolarity := 23,
	eEngineeringUnits := 25,
	ePriorityValue := 26,
	eLimitEnable := 27,
	eNotifyType := 29,
	eTimeStamp := 30,
	eDeviceObjectPropertyReference := 31,
	eDeviceStatus := 32,
	eServicesSupported := 33,
	eObjectTypesSupported := 34,
	eSegmentation := 35,
	eVTClass := 36,
	eVTSession := 37,
	eSessionKey := 38,
	eRecipient := 39,
	eAddressBinding := 40,
	eCOVSubscription := 41,
	eEventType := 42,
	eEventParameter := 43,
	eFileAccessMethod := 44,
	eReadAccessSpecification := 45,
	eReadAccessResult := 46,
	eObjectPropertyReference := 47,
	eSetpointReference := 48,
	eDestination := 49,
	eProgramState := 50,
	eProgramRequest := 51,
	eProgramError := 52,
	eDateRange := 53,
	eDailySchedule := 54,
	eSpecialEvent := 55,
	eClientCOV := 56,
	eLogRecord := 57,
	eLifeSafetyState := 58,
	eLifeSafetyMode := 59,
	eSilencedState := 60,
	eLifeSafetyOperation := 61,
	eBinaryPV := 62,
	eDaysOfWeek := 63,
	eWeekNDay := 64,
	eTimeValue := 65,
	eValue := 66,
	eAddress := 67,
	ePropertyIdentifier := 68,
	eEnumerationValueType := 69,
	eBitFieldBit := 70,
	eLogDatum := 71,
	eAnyType := 72,
	ePresentValue := 73,
	eContextTag := 74,
	eValueChoice := 75,
	eLogStatus := 76,
	eRecipientProcess := 77,
	eSubscribeCOVPropertyRequest := 78,
	ePropertyReference := 79,
	ePropertyResult := 80,
	eDeviceObjectPropertyValue := 81,
	eCOVNotificationRequest := 82,
	eEventNotificationRequest := 83,
	eNotificationParameters := 84,
	eChangeOfBitstring := 85,
	eChangeOfState := 86,
	eChangeOfValue := 87,
	eCommandFailure := 88,
	eFloatingLimit := 89,
	eOutOfRange := 90,
	ePropertyValue := 91,
	eComplexTag := 92,
	eChangeOfLifeSafety := 93,
	eExtended := 94,
	eBufferReady := 95,
	eUnsignedRange := 96,
	ePropertyResultValue := 97,
	eServiceCOVPropSubscription := 98,
	eServiceCOVSubscription := 99,
	eCOVNotification := 100,
	eAcknowledgeAlarmRequest := 101,
	eVTOpenRequest := 102,
	ePrescale := 103,
	eScale := 104,
	eAction := 105,
	eError := 106,
	eErrorType := 107,
	eErrorClass := 108,
	eErrorCode := 109,
	eRejectReason := 110,
	eAbortReason := 111,
	eBDTEntry := 112,
	eIpEntry := 113,
	eMaskEntry := 114,
	eEthernetAddress := 115,
	eLonTalkAddress := 116,
	eLonTalkNeuronId := 117,
	eNodeType := 118,
	eDeviceObjectReference := 119,
	eActionCommand := 120,
	eGetEventInformation := 121,
	eGetEnrollmentSummaryCriteria := 122,
	eGetEnrollmentSummaryCriteriaResponse := 123,
	eDeviceCommunicationControl := 124,
	eInt16 := 125,
	eUInt16 := 126,
	eUInt8 := 127,
	eTypeInt8 := 128,
	eByte := 129,
	eFDTEntry := 130,
	eAddress_3 := 131,
	eAddress_4 := 132,
	eAddress_5 := 133,
	ePersistentDataState := 134,
	eFallbackRealValue := 135,
	eFallbackBinaryValue := 136,
	eRealNull := 137,						// PresentValue in AnalogObj
	eEnumeratedNull := 138,					// PresentValue in BinaryObj
	eUnsignedIntegerNull := 139,			// PresentValue in Multistate
	eUnknown := 140,
	eDiagnosisPerformance := 200,
	eDiagnosisEthStatistics := 201,
	eFrameStatistics := 202,
	eInfo := 203,
	eDiagnosis := 204,
	eTcIoEthStatistic := 205,
	eTcIoEthTxRxErrorCount := 206,
	eTcIoEthPortStatistic := 207,
	eServerStatistics := 208,
	eFrameServicesDiag := 209,
	eUnsignedIntegerArr := 258,
	eCharacterStringExtArr := 263,
	eObjectIdentifierArr := 268,
	eCalendarEntryArr := 272,
	eActionListArr := 275,
	ePriorityValueArr := 282,
	eTimeStampArr := 286,
	eDeviceObjectPropertyReferenceArr := 287,
	eVTClassArr := 292,
	eVTSessionArr := 293,
	eSessionKeyArr := 294,
	eRecipientArr := 295,
	eAddressBindingArr := 296,
	eCOVSubscriptionArr := 297,
	eReadAccessSpecificationArr := 301,
	eReadAccessResultArr := 302,
	eDestinationArr := 305,
	eSpecialEventArr := 311,
	eLogRecordArr := 313,
	eLifeSafetyStateArr := 314,
	eTimeValueArr := 321,
	eUnsignedIntegerList := 514,
	eCharacterStringExtList := 519,
	eReadAccessSpecificationList := 557,
	eReadAccessResultList := 558,
	eSpecialEventList := 567,
	eLogRecordList := 569,
	eTimeValueList := 577,
	eValueList := 578,
	eLogDatumList := 583,
	ePropertyReferenceList := 591,
	ePropertyResultList := 592,
	eCOVNotificationRequestList := 594,
	eEventNotificationRequestList := 595,
	ePropertyValueList := 603,
	eDailyScheduleList := 1089
);
END_TYPE

// DUTs/Enumerations/Properties/E_BACnet_DeviceStatus
{attribute 'qualified_only'}
TYPE E_BACnet_DeviceStatus:
(
	Invalid					:= -1,
	
	eOperational 			:= 0,
	eOperationalReadOnly	:= 1,
	eDownloadRequired 		:= 2,
	eDownloadInProgress 	:= 3,
	eNonOperational 		:= 4,
	eBackupInProgress 		:= 5
);
END_TYPE

// DUTs/Enumerations/Properties/E_BACnet_FileAccessMethod
{attribute 'qualified_only'}
TYPE E_BACnet_FileAccessMethod:
(
	Invalid := -1,
	
	eRecordAccess := 0,
	eStreamAccess := 1
);
END_TYPE

// DUTs/Enumerations/Properties/E_BACnet_LifeSafetyMode
{attribute 'qualified_only'}
TYPE E_BACnet_LifeSafetyMode:
(
	Invalid := -1,
	
	eOff := 0,
	eOn := 1,
	eTest := 2,
	eManned := 3,
	eUnmanned := 4,
	eArmed := 5,
	eDisarmed := 6,
	ePrearmed := 7,
	eSlow := 8,
	eFast := 9,
	eDisconnected := 10,
	eEnabled := 11,
	eModeDisabled := 12,
	eAutomaticReleaseDisabled := 13,
	eModeDefault := 14
);
END_TYPE

// DUTs/Enumerations/Properties/E_BACnet_LifeSafetyOperation
{attribute 'qualified_only'}
TYPE E_BACnet_LifeSafetyOperation:
(
	Invalid := -1,
	
	eNone := 0,
	eSilence := 1,
	eSilenceAnble := 2,
	eSilenceVisual := 3,
	eReset := 4,
	eResetAlarm := 5,
	eResetFault := 6,
	eUnsilence := 7,
	eUnsilenceAnble := 8,
	eUnsilenceVisual := 9
);
END_TYPE

// DUTs/Enumerations/Properties/E_BACnet_LimitEnableBits
{attribute 'qualified_only'}
TYPE E_BACnet_LimitEnableBits:
(
	Invalid := -1,
	
	eLowLimit := 0,
	eHighLimit := 1
);
END_TYPE

// DUTs/Enumerations/Properties/E_BACnet_LoopMode
{attribute 'qualified_only'}
TYPE E_BACnet_LoopMode :
(
	Invalid := -1,
	
	eNone,					// LOOP object has unknown parameter settings
	eIdeal,					// Controller is in ideal form: P, I and D are in parallel junktion; unit of P, I and D is [1] (Kp, Ki, Kd)
	eStandard				// Controller works in standard form (most industrial applications): P parameter is applied to I and D; unit of I and D is time based [s] (Kp, Ti, Td)
);
END_TYPE

// DUTs/Enumerations/Properties/E_BACnet_NodeType
{attribute 'qualified_only'}
TYPE E_BACnet_NodeType :
(
	Invalid := -1,
	
	eUnknown := 0,
	eSystem := 1,
	eNetwork := 2,
	eDevice := 3,
	eOrganizational := 4,
	eArea := 5,
	eEquipment := 6,
	ePoint := 7,
	eCollection := 8,
	eProperty := 9,
	eFunctional := 10,
	eOther := 11
);
END_TYPE

// DUTs/Enumerations/Properties/E_BACnet_NotifyType
{attribute 'qualified_only'}
TYPE E_BACnet_NotifyType:
(
	Invalid				:= -1,
	
	eAlarm				:= 0,
	eNotifyEvent		:= 1
//	ntAckNotification	:= 2
);
END_TYPE

// DUTs/Enumerations/Properties/E_BACnet_ObjectSupportedBits
{attribute 'qualified_only'}
TYPE E_BACnet_ObjectSupportedBits:
(
	Invalid := -1,
	
	eAnalogInput := 0,
	eAnalogOutput := 1,
	eAnalogValue := 2,
	eBinaryInput := 3,
	eBinaryOutput := 4,
	eBinaryValue := 5,
	eCalendar := 6,
	eCommand := 7,
	eDevice := 8,
	eEventEnrollment := 9,
	eFile := 10,
	eGroup := 11,
	eLoop := 12,
	eMultiStateInput := 13,
	eMultiStateOutput := 14,
	eNotificationClass := 15,
	eProgr := 16,
	eSchedule := 17,
	eAveraging := 18,
	eMultiStateValue := 19,
	eTrendLog := 20,
	eLifeSafetyPoint := 21,
	eLifeSafetyZone := 22,
	eAccumulator := 23,
	ePulseConverter := 24,
	eEventLog := 25,
	eGlobalGroup := 26,
	eTrendLogMultiple := 27,
	eLoadControl := 28,
	eStructuredView := 29,
	eAccessDoor := 30,
	eunassigend31 := 31,
	eAccessCredential := 32,
	eAccessPoint := 33,
	eAccessRights := 34,
	eAccessUser := 35,
	eAccessZone := 36,
	eCredentialDataInput := 37,
	eNetworkSecurity := 38,
	eBitStringValue := 39,
	eCharacterStringValue := 40,
	eDatePatternValue := 41,
	eDateValue := 42,
	eDateTimePatternValue := 43,
	eDateTimeValue := 44,
	eIntegerValue := 45,
	eLargeAnalogValue := 46,
	eOctetStringValue := 47,
	ePositiveIntegerValue := 48,
	eTimePatternValue := 49,
	eTimeValue := 50,
	eNetworkPort := 51,
	eAlertEnrollment := 52,
	eChannel := 53
);
END_TYPE

// DUTs/Enumerations/Properties/E_BACnet_PersistentDataState
{attribute 'qualified_only'}
TYPE E_BACnet_PersistentDataState :
(
	Invalid			:= -1,
	
	eDisabled		:= 0,
	eInitialize		:= 1,
	eNoChange		:= 2,
	eReady			:= 3,
	eWrite			:= 4,
	eWriting		:= 5
);
END_TYPE

// DUTs/Enumerations/Properties/E_BACnet_Priority
{attribute 'qualified_only'}
{warning disable C0125}
TYPE E_BACnet_Priority:
(
	Invalid			:= -1,
	
	eP1				:= 1,
	eP2				:= 2,
	eP3				:= 3,
	eP4				:= 4,
	eP5				:= 5,
	eP6				:= 6,
	eP7				:= 7,
	eP8				:= 8,
	eP9				:= 9,
	eP10			:= 10,
	eP11			:= 11,
	eP12			:= 12,
	eP13			:= 13,
	eP14			:= 14,
	eP15			:= 15,
	eP16			:= 16,
	
	eDefault		:= 17,
	
	First			:= eP1,
	Last			:= eP16,
	Count			:= (Last - First + 1)
);
END_TYPE
{warning restore C0125}

// DUTs/Enumerations/Properties/E_BACnet_ProgramError
{attribute 'qualified_only'}
TYPE E_BACnet_ProgramError:
(
	Invalid				:= -1,
	
	eProgramNormal		:= 0,
	eLoadFailed			:= 1,
	eProgerrorInternal	:= 2,
	eProgram			:= 3,
	eOther				:= 4
);
END_TYPE

// DUTs/Enumerations/Properties/E_BACnet_ProgramRequest
{attribute 'qualified_only'}
TYPE E_BACnet_ProgramRequest:
(
	Invalid		:= -1,
	
	eReady		:= 0,
	eLoad		:= 1,
	eRun		:= 2,
	eHalt		:= 3,
	eRestart	:= 4,
	eUnload		:= 5
);
END_TYPE

// DUTs/Enumerations/Properties/E_BACnet_ProgramState
{attribute 'qualified_only'}
TYPE E_BACnet_ProgramState:
(
	Invalid			:= -1,
	
	eIdle			:= 0,
	eLoading		:= 1,
	eRunning		:= 2,
	eWaiting		:= 3,
	eHalted			:= 4,
	eUnloading		:= 5
);
END_TYPE

// DUTs/Enumerations/Properties/E_BACnet_RejectReason
{attribute 'qualified_only'}
{warning disable C0125}
TYPE E_BACnet_RejectReason :
(
	Invalid							:= -1,
	
	eOther							:= 0,
	eBufferOverflow					:= 1,
	eInconsistentParameters			:= 2,
	eInvalidParameterDataType		:= 3,
	eInvalidTag						:= 4,
	eMissingRequiredParameter		:= 5,
	eParameterOutOfRange			:= 6,
	eTooManyArguments				:= 7,
	eUndefinedEnumeration			:= 8,
	eUnrecognizedService			:= 9,
	
	NoReason						:= 256,
	First							:= eOther,
	Last							:= eUnrecognizedService,
	Count							:= (Last - First + 1)
);
END_TYPE
{warning restore C0125}

// DUTs/Enumerations/Properties/E_BACnet_RestartReason
{attribute 'qualified_only'}
{attribute 'strict'}
TYPE E_BACnet_RestartReason :
(
	Invalid						:= -1,
	
	eReasonUnknown				:= 0,
	eReasonColdstart			:= 1,
	eReasonWarmstart			:= 2,
	eReasonDetectPowerLost		:= 3,
	eReasonDetectPowerOff		:= 4,
	eReasonHardwareWatchdog		:= 5,
	eReasonSoftwareWatchdog		:= 6,
	eReasonSuspended			:= 7
);
END_TYPE

// DUTs/Enumerations/Properties/E_BACnet_ScaleChoice
{attribute 'qualified_only'}
{attribute 'strict'}
TYPE E_BACnet_ScaleChoice :
(
	Invalid			:= -1,
	
	eFloatScale		:= 0,
	eIntegerScale	:= 1
);
END_TYPE

// DUTs/Enumerations/Properties/E_BACnet_Segmentation
{attribute 'qualified_only'}
TYPE E_BACnet_Segmentation:
(
	Invalid		:= -1,
	
	eBoth		:= 0,
	eTransmit	:= 1,
	eReceive	:= 2,
	eNo			:= 3
);
END_TYPE

// DUTs/Enumerations/Properties/E_BACnet_ServicesSupportedBits
{attribute 'qualified_only'}
TYPE E_BACnet_ServicesSupportedBits:
(
	eSuppInvalid := -1,
	
	eSuppAcknowledgeAlarm := 0,
	eSuppConfirmedCOVNotification := 1,
	eSuppConfirmedEventNotification := 2,
	eSuppGetAlarmSummary := 3,
	eSuppGetEnrollmentSummary := 4,
	eSuppSubscribeCOV := 5,
	eSuppAtomicReadFile := 6,
	eSuppAtomicWriteFile := 7,
	eSuppAddListElement := 8,
	eSuppRemoveListElement := 9,
	eSuppCreateObject := 10,
	eSuppDeleteObject := 11,
	eSuppReadProperty := 12,
	eSuppReadPropertyConditional := 13,
	eSuppReadPropertyMultiple := 14,
	eSuppWriteProperty := 15,
	eSuppWritePropertyMultiple := 16,
	eSuppDeviceCommunicationControl := 17,
	eSuppConfirmedPrivateTransfer := 18,
	eSuppConfirmedTextMessage := 19,
	eSuppReinitializeDevice := 20,
	eSuppVtOpen := 21,
	eSuppVtClose := 22,
	eSuppVtData := 23,
	eSuppAuthenticate := 24,
	eSuppRequestKey := 25,
	eSuppIAm := 26,
	eSuppIHave := 27,
	eSuppUnconfirmedCOVNotification := 28,
	eSuppUnconfirmedEventNotification := 29,
	eSuppUnconfirmedPrivateTransfer := 30,
	eSuppUnconfirmedTextMessage := 31,
	eSuppTimeSynchronization := 32,
	eSuppWhoHas := 33,
	eSuppWhoIs := 34,
	eSuppReadRange := 35,
	eSuppUtcTimeSynchronization := 36,
	eSuppLifeSafetyOperation := 37,
	eSuppSubscribeCOVProperty := 38,
	eSuppGetEventInformation := 39
);
END_TYPE

// DUTs/Enumerations/Properties/E_BACnet_SilencedState
{attribute 'qualified_only'}
TYPE E_BACnet_SilencedState:
(
	Invalid				:= -1,
	
	eUnsilenced			:= 0,
	eAnbleSilenced		:= 1,
	eVisibleSilenced	:= 2,
	eAllSilenced		:= 3
);
END_TYPE

// DUTs/Enumerations/Properties/E_BACnet_StatusFlags
{attribute 'qualified_only'}
TYPE E_BACnet_StatusFlags:
(
	Invalid			:= -1,
	
	eInAlarm		:= 0,
	eFault			:= 1,
	eOverridden		:= 2,
	eOutOfService	:= 3
);
END_TYPE

// DUTs/Enumerations/Properties/E_BACnet_StringEncodingTypes
{attribute 'qualified_only'}
TYPE E_BACnet_StringEncodingTypes :
(
	Invalid		:= -1,
	
	eAnsiUTF8	:= 0,
	eDBCS		:= 1,
	eJIS		:= 2,
	eUCS4		:= 3,
	eUCS2		:= 4,
	eISO8859	:= 5
);
END_TYPE

(*
---------------------------------------------
ISO8859
---------------------------------------------
						Part 1	Latin-1_ Western European__					
						Part 2	Latin-2_ Central European__					
						Part 3	Latin-3_ South European__					
						Part 4	Latin-4_ North European__					
Part 5	Latin/Cyrillic
Part 6	Latin/Arabic
Part 7	Latin/Greek
Part 8	Latin/Hebrew
						Part 9	Latin-5 _Turkish__					
						Part 10	Latin-6 _Nordic__					
Part 11	Latin/Thai
Part 12	"non-existent part" Latin/Devanagari
						Part 13	Latin-7_ Baltic Rim__					
						Part 14	Latin-8_ Celtic__					
Part 15	Latin-9
						Part 16	Latin-10_ South-Eastern European__					
---------------------------------------------
*)

// DUTs/Enumerations/Remote/E_BACnetRM_ClientState
{attribute 'qualified_only'}
TYPE E_BACnetRM_ClientState :
(
	eInit,
	eReadSupportedServices,
	eCalcAuto,
	eReadApduSize,
	eCreateRequests,
	eCycle,
	eReInit,
	eError
);
END_TYPE

// DUTs/Enumerations/Remote/E_BACnetRM_RequestType
{attribute 'qualified_only'}
TYPE E_BACnetRM_RequestType :
(
	eUndefined,
	
	eRead,
	eReadPropertyMultiple,
	eWrite,
	eWritePropertyMultiple,
	eCOV,
	eCOV_C,
	eCOV_U,
	eAcknowledge,
	eAddListElement,
	eRemoveListElement
);
END_TYPE

// DUTs/Enumerations/E_BACnet_Error
{attribute 'qualified_only'}
{warning disable C0125}
TYPE E_BACnet_Error :
(
	eNoError														:= 0,
	
	// General:
	eNoValidNetId													:= 1,
	eWrongMapping													:= 2,
	eOperational													:= 3,
	eNoEthLink														:= 4,
	eNoGateway														:= 5,
	eWocTriggerUnsup												:= 6,
	eWocDisabled													:= 7,
	eInvalidObjectId												:= 8,
	eInvalidObjectType												:= 10,
	eInvalidCycleTime												:= 11,
	eInvalidParameter												:= 12,
	eInvalidClient													:= 14,
	eInvalidServer													:= 15,
	eNotFoundBySymbol												:= 16,
	eCreateObject													:= 17,
	eDeviceNotFound													:= 18,
	eDuplicateObjectId												:= 19,

	// Errors with reset:
	ePersistentWrite												:= 20,
	eInvalidAdsConn													:= 21,
	eClientTimeout													:= 22,
	eClientService													:= 23,
	eWocTriggerActive												:= 24,
	eRevisionRead													:= 25,
	ePersistentPlcWrite												:= 26,
	eInvalidTask													:= 27,

	// ADS connection errors:
	eADS_NoValidNetId												:= 30,						// missing a valid Net ID
	eADS_Data														:= 31,						// ADS data length is wrong
	eADS_Read														:= 32,						// ADS read function was aborted
	eADS_Write														:= 33,						// ADS write function was aborted
	eADS_ObjType													:= 34,						// object type is wrong
	eADS_ObjListEmpty												:= 35,						// object list is empty
	eADS_DeviceOp													:= 36,						// device is not operational
	eADS_NoDevice													:= 37,						// no device object in object info list
	eADS_ObjInstance												:= 38,						// object list info is wrong
	eADS_AmsPort													:= 39,						// read AMS port is invalid (<1000)
	eADS_ObjectId													:= 40,						// object list info is wrong
	eADS_LegacyStack												:= 41,						// revision 6 stack detected (service is available from/above revision 9)
	eADS_ObjIdMissmatch												:= 42,						// object ID mapped and object list info are different
	eADS_BufferSize													:= 43,						// Property data larger than ADS buffer
	eADS_SchedData													:= 44,						// Wrong schedule property data
	eUnknownEventChoice												:= 45,						// Unknown event choice type
	eUnknownEntryChoice												:= 46,						// Unknown entry choice type
	eADS_TooManyObjects												:= 47,						// List of objects are longer than output list size
	eADS_WrongEntrySize												:= 48,						// expected entry size dosn't match read size
	eADS_RecipientData												:= 49,						// Invalid recipient data, device type expected
	eADS_TooManyEntries												:= 50,						// More entries than expected
	eADS_NotEnoughEntries											:= 51,						// Property incomplete, missing entries
	eADS_Encoding													:= 52,						// String encoding not supported
	eADS_NoServerClient												:= 53,						// Given ADS connection is not an server or client connection (expected bClient or bServer)
	eADS_NoNotificationSink											:= 54,						// Given ADS connection is not an notification sink connection (expected bNSink)
	
	FirstResetError													:= ePersistentWrite,
	LastResetError													:= eInvalidTask
);
END_TYPE
{warning restore C0125}

// DUTs/Types/[ADS]/ST_BACnet_AdsConnection
{attribute 'hide'}
TYPE ST_BACnet_AdsConnection :
STRUCT
	bValid		: BOOL; (* information are valid *)
	nReload		: USINT; (* reload counter *)
	sAmsNetId	: T_AmsNetId;
	nAmsPort	: T_AmsPort := 1000;
	bServer		: BOOL;
	bClient		: BOOL;
	bNSink		: BOOL;
	nDeviceId	: UDINT; (* Device object instance resp. BACnet ID *)
END_STRUCT
END_TYPE

// DUTs/Types/[Functional]/U_BACnet_CreateObj
{attribute 'hide'}
TYPE U_BACnet_CreateObj :
UNION
	Obj			: POINTER TO FB_BACnet_Object;
	
	AIRaw		: POINTER TO FB_BACnet_AI_Raw;
	AORaw		: POINTER TO FB_BACnet_AO_Raw;
	AORaw5P		: POINTER TO FB_BACnet_AO_Raw5P;
	AV			: POINTER TO FB_BACnet_AV;
	AV5P		: POINTER TO FB_BACnet_AV_5P;
	AVDisp		: POINTER TO FB_BACnet_AV_Disp;
	AVSetp		: POINTER TO FB_BACnet_AV_Setp;
	
	BIRaw		: POINTER TO FB_BACnet_BI_Raw;
	BORaw		: POINTER TO FB_BACnet_BO_Raw;
	BORaw5P		: POINTER TO FB_BACnet_BO_Raw5P;
	BV			: POINTER TO FB_BACnet_BV;
	BV5P		: POINTER TO FB_BACnet_BV_5P;
	BVDisp		: POINTER TO FB_BACnet_BV_Disp;
	BVSetp		: POINTER TO FB_BACnet_BV_Setp;
	
	MIRaw		: POINTER TO FB_BACnet_MI_Raw;
	MORaw		: POINTER TO FB_BACnet_MO_Raw;
	MORaw5P		: POINTER TO FB_BACnet_MO_Raw5P;
	MV			: POINTER TO FB_BACnet_MV;
	MV5P		: POINTER TO FB_BACnet_MV_5P;
	MVDisp		: POINTER TO FB_BACnet_MV_Disp;
	MVSetp		: POINTER TO FB_BACnet_MV_Setp;
	
	Clnd		: POINTER TO FB_BACnet_Cal;
	Device		: POINTER TO FB_BACnet_Device;
	File		: POINTER TO FB_BACnet_File;
	Loop		: POINTER TO FB_BACnet_Loop;
	NC			: POINTER TO FB_BACnet_NC;
	Prog		: POINTER TO FB_BACnet_Prog;
	SchedA		: POINTER TO FB_BACnet_SchedA;
	SchedB		: POINTER TO FB_BACnet_SchedB;
	SchedM		: POINTER TO FB_BACnet_SchedM;
	Acc			: POINTER TO FB_BACnet_Acc;
	PC			: POINTER TO FB_BACnet_PC;
	View		: POINTER TO FB_BACnet_View;
	
END_UNION
END_TYPE

// DUTs/Types/Diagnose/ST_BACnet_ConfirmedServiceDiag
{attribute 'hide'}
TYPE ST_BACnet_ConfirmedServiceDiag :
STRUCT
	nReqSend: DWORD; (* ULONG *)
	nReqSendFail: DWORD; (* ULONG *)
	nReqRecv: DWORD; (* ULONG *)
	nReqRecvFail: DWORD; (* ULONG *)
	nAckSend: DWORD; (* ULONG *)
	nAckSendFail: DWORD; (* ULONG *)
	nAckRecv: DWORD; (* ULONG *)
	nAckRecvFail: DWORD; (* ULONG *)
END_STRUCT
END_TYPE

// DUTs/Types/Diagnose/ST_BACnet_DiagEthStatistics
{attribute 'hide'}
TYPE ST_BACnet_DiagEthStatistics :
STRUCT
	ethStat: ST_BACnet_TcIoEthStatistic;
	txRxErrCnt: ST_BACnet_TcIoEthTxRxErrorCount;
END_STRUCT
END_TYPE

// DUTs/Types/Diagnose/ST_BACnet_Diagnosis
{attribute 'hide'}
TYPE ST_BACnet_Diagnosis :
STRUCT
	ethDevice: ST_BACnet_DiagEthStatistics;
	execTiming: ST_BACnet_DiagnosisTiming;
	frameStatistics: ST_BACnet_FrameStatistics;
	nRes1 : DWORD;
	info: ST_BACnet_Info;
	nRes2 : DWORD;
	serverInfo: ST_BACnet_ServerStatistics;
	lastUpdate: ST_BA_DateTime;
	nRes3 : DWORD;
END_STRUCT
END_TYPE

// DUTs/Types/Diagnose/ST_BACnet_DiagnosisTiming
{attribute 'hide'}
TYPE ST_BACnet_DiagnosisTiming :
STRUCT
	msIoInCurExecutionTime: DWORD; (* ULONG *)
	msIoInMinExecutionTime: DWORD; (* ULONG *)
	msIoInMaxExecutionTime: DWORD; (* ULONG *)
	msIoOutCurExecutionTime: DWORD; (* ULONG *)
	msIoOutMinExecutionTime: DWORD; (* ULONG *)
	msIoOutMaxExecutionTime: DWORD; (* ULONG *)
	msCycleCurExecutionTime: DWORD; (* ULONG *)
	msCycleMinExecutionTime: DWORD; (* ULONG *)
	msCycleMaxExecutionTime: DWORD; (* ULONG *)
	msInputCurDistanceTime: DWORD; (* ULONG *)
	msInputMinDistanceTime: DWORD; (* ULONG *)
	msInputMaxDistanceTime: DWORD; (* ULONG *)
END_STRUCT
END_TYPE

// DUTs/Types/Diagnose/ST_BACnet_FrameStatistics
{attribute 'hide'}
TYPE ST_BACnet_FrameStatistics :
STRUCT
	confirmed: ARRAY[0..29] OF ST_BACnet_ConfirmedServiceDiag; (* [SERVICE_CONFIRMED_MAX + 1]; 29 + 1 *)
	unConfirmed: ARRAY[0..9] OF ST_BACnet_UnConfirmedServiceDiag; (* [SERVICE_UNCONFIRMED_MAX + 1]; 9 *)
	nSegmSendTimeouts: DWORD; (* ULONG *)
	nFrameAllocFailCnt: DWORD; (* ULONG *)
	nFrameSendCnt: DWORD; (* ULONG *)
	nFrameSendFailCnt: DWORD; (* ULONG *)
	nFrameRecvCnt: DWORD; (* ULONG *)
	nFrameRecvFailCnt: DWORD; (* ULONG *)
	nLinkStatusChangedCnt: DWORD; (* ULONG *)
END_STRUCT
END_TYPE

// DUTs/Types/Diagnose/ST_BACnet_Info
{attribute 'hide'}
TYPE ST_BACnet_Info :
STRUCT
	nAmsAllocCnt: DINT; (* LONG *)
	nAmsAllocCntMax: DWORD; (* ULONG *)
	nAmsAllocFailCnt: DWORD; (* ULONG *)
	nAvailPhysMemBytes: DWORD; (* ULONG *)
	nAvailFlashMemBytes: ARRAY[0..1] OF DWORD; (* ULONGLONG *)
	nRecvFrameFifoSize: DWORD; (* ULONG *)
	nEmptyFrameFifoSize: DWORD; (* ULONG *)
	nRecvSegmUDPFramesListSize: DWORD; (* ULONG *)
	nRecvSegmFramesListSize: DWORD; (* ULONG *)
	nSendSegmFramesListSize: DWORD; (* ULONG *)
	nClientScanListSize: DWORD; (* ULONG *)
	nAmsRecvMissCount: DWORD; (* ULONG *)
END_STRUCT
END_TYPE

// DUTs/Types/Diagnose/ST_BACnet_ServerStatistics
{attribute 'hide'}
TYPE ST_BACnet_ServerStatistics :
STRUCT
	nOpenRequests: DWORD; (* ULONG *)
	nRequestRetries: DWORD; (* ULONG *)
	nRequestTimeOuts: DWORD; (* ULONG *)
	nPropChanges: DWORD; (* ULONG *)
	nPersistWrites: DWORD; (* ULONG *)
	persistChangeSetId: DWORD; (* ULONG *)
	secpersistNextWrite: DWORD; (* ULONG *)
	persistLastWrite: ST_BA_DateTime;
END_STRUCT
END_TYPE

// DUTs/Types/Diagnose/ST_BACnet_TcIoEthStatistic
{attribute 'hide'}
TYPE ST_BACnet_TcIoEthStatistic :
STRUCT
	dcTimeStamp: ARRAY[0..1] OF DWORD; (* ULONGLONG *)
	sendFrames: DWORD; (* ULONG *)
	recvFrames: DWORD; (* ULONG *)
	sendTimeRTime: DWORD; (* ULONG *)
	recvTimeRTime: DWORD; (* ULONG *)
	sendTimeNdis: DWORD; (* ULONG *)
	recvTimeNdis: DWORD; (* ULONG *)
END_STRUCT
END_TYPE

// DUTs/Types/Diagnose/ST_BACnet_TcIoEthTxRxErrorCount
{attribute 'hide'}
TYPE ST_BACnet_TcIoEthTxRxErrorCount :
STRUCT
	txCnt: DWORD; (* ULONG *)
	rxCnt: DWORD; (* ULONG *)
END_STRUCT
END_TYPE

// DUTs/Types/Diagnose/ST_BACnet_UnConfirmedServiceDiag
{attribute 'hide'}
TYPE ST_BACnet_UnConfirmedServiceDiag :
STRUCT
	nReqSend: DWORD; (* ULONG *)
	nReqSendFail: DWORD; (* ULONG *)
	nReqRecv: DWORD; (* ULONG *)
	nReqRecvFail: DWORD; (* ULONG *)
END_STRUCT
END_TYPE

// DUTs/Types/Properties/[ADS]/Calendar/ST_BACnet_CalendarEntry
TYPE ST_BACnet_CalendarEntry :
STRUCT
	eEventChoice		: E_BACnet_CalendarEntryChoice;
	{attribute 'hide'}
	_res1				: UINT;
	uCalEntry			: U_BA_DateVal;
END_STRUCT
END_TYPE

// DUTs/Types/Properties/[ADS]/Calendar/ST_BACnet_CalendarEntryDate
{attribute 'hide'}
TYPE ST_BACnet_CalendarEntryDate :
STRUCT
(*
	typedef struct _BACnetCalendarEntry
	{
	      BACnetCalendarEntryChoice choice;
	      union
	      {
	            BACnetDate              date;
	            BACnetDateRange   dateRange;
	            BACnetWeekNDay          weekNDay;
	      };
	}BACnetCalendarEntry, *PBACnetCalendarEntry;
*)
	eEntryChoice		: E_BACnet_CalendarEntryChoice;
	nRes				: WORD; (* ENUM alignment *)
	stDate				: ST_BA_Date;
END_STRUCT
END_TYPE

// DUTs/Types/Properties/[ADS]/Calendar/ST_BACnet_CalendarEntryDateRange
{attribute 'hide'}
TYPE ST_BACnet_CalendarEntryDateRange :
STRUCT
(*
	typedef struct _BACnetCalendarEntry
	{
	      BACnetCalendarEntryChoice choice;
	      union
	      {
	            BACnetDate              date;
	            BACnetDateRange   dateRange;
	            BACnetWeekNDay          weekNDay;
	      };
	}BACnetCalendarEntry, *PBACnetCalendarEntry;
*)
	eEntryChoice		: E_BACnet_CalendarEntryChoice;
	nRes				: WORD; (* ENUM alignment *)
	stStartDate			: ST_BA_Date;
	stEndDate			: ST_BA_Date;
END_STRUCT
END_TYPE

// DUTs/Types/Properties/[ADS]/Calendar/ST_BACnet_CalendarEntryWeekNDay
{attribute 'hide'}
TYPE ST_BACnet_CalendarEntryWeekNDay :
STRUCT
(*
	typedef struct _BACnetCalendarEntry
	{
	      BACnetCalendarEntryChoice choice;
	      union
	      {
	            BACnetDate              date;
	            BACnetDateRange   dateRange;
	            BACnetWeekNDay          weekNDay;
	      };
	}BACnetCalendarEntry, *PBACnetCalendarEntry;
*)
	eEntryChoice	: E_BACnet_CalendarEntryChoice;
	nRes1			: WORD; (* ENUM alignment *)
	nMonth			: USINT;
	nWeekOfMonth	: USINT;
	nDay			: USINT;
	nRes2			: USINT; (* weekNDay alignment *)
END_STRUCT
END_TYPE

// DUTs/Types/Properties/[ADS]/Calendar/T_BACnet_CalendarEntryTypeFilter
{attribute 'hide'}
TYPE T_BACnet_CalendarEntryTypeFilter : ARRAY[0..4] OF E_BACnet_CalendarEntryType; END_TYPE

// DUTs/Types/Properties/[ADS]/DateTime/ST_BACnet_TimeStampDateTime
{attribute 'hide'}
TYPE ST_BACnet_TimeStampDateTime :
STRUCT
	eType		: E_BACnet_TimeStampChoice := E_BACnet_TimeStampChoice.eDateTime;
	{attribute 'hide'}
	nReserve1	: WORD;
	stDateTime	: ST_BA_DateTime;
END_STRUCT
END_TYPE

// DUTs/Types/Properties/[ADS]/DateTime/ST_BACnet_TimeValue
{attribute 'hide'}
TYPE ST_BACnet_TimeValue :
STRUCT
	stTime	: ST_BA_Time;
	nRes	: DWORD;
	stValue	: ST_BACnet_Value;
END_STRUCT
END_TYPE

// DUTs/Types/Properties/[ADS]/DateTime/ST_BACnet_TimeValueBool
{attribute 'hide'}
TYPE ST_BACnet_TimeValueBool :
STRUCT
	bValid		: BOOL;
	stTime		: ST_BA_Time;
	eType		: E_BACnet_DataTypes;
	bValue		: BOOL;
END_STRUCT
END_TYPE

// DUTs/Types/Properties/[ADS]/DateTime/ST_BACnet_TimeValueList
{attribute 'hide'}
TYPE ST_BACnet_TimeValueList :
STRUCT
	nEntrySize	: DWORD;
	nRes		: DWORD;
	stListEntry	: ST_BACnet_TimeValue;
END_STRUCT
END_TYPE

// DUTs/Types/Properties/[ADS]/DateTime/ST_BACnet_TimeValueReal
{attribute 'hide'}
TYPE ST_BACnet_TimeValueReal :
STRUCT
	bValid		: BOOL;
	stTime		: ST_BA_Time;
	eType		: E_BACnet_DataTypes;
	fValue		: REAL;
END_STRUCT
END_TYPE

// DUTs/Types/Properties/[ADS]/LogBuffer/ST_BACnet_LogBufferEntryReal
{attribute 'hide'}
TYPE ST_BACnet_LogBufferEntryReal :
STRUCT
	nTimeStamp	: DWORD; (* 100ms since 1900 *)
	stDateTime	: ST_BA_DateTime; (* BACnet time stamp *)
	fValue		: REAL;
END_STRUCT
END_TYPE

// DUTs/Types/Properties/[ADS]/LogBuffer/ST_BACnet_LogBufferReal
{attribute 'hide'}
TYPE ST_BACnet_LogBufferReal :
STRUCT
	nGet		: USINT; (* Update date counter *)
	sObjectDesc	: T_MAXSTRING; (* Object description *)
	nCount		: UDINT; (* log buffer entries *)
	arrEntries	: ARRAY[0..BACnet_Globals.nDataField_MaxLogBufferEntries] OF ST_BACnet_LogBufferEntryReal;
END_STRUCT
END_TYPE

// DUTs/Types/Properties/[ADS]/LogRecord/ST_BACnet_LogDatum
{attribute 'hide'}
TYPE ST_BACnet_LogDatum :
STRUCT
(*

typedef struct _BACnetLogDatum
{
      BACnetLogRecordChoice choice;
      union
      {
            DWORD logStatus; // BitString ... of type BACnetLogStatus
            BOOL booleanValue;
            FLOAT realValue;
            EnumerationValueType enumerationValue;
            ULONG unsignedValue;
            DWORD signedValue;
            DWORD bitstringValue;
            DWORD nullValue;
            BACnetError failure; 
            FLOAT timeChange;
            AnyType anyValue; // ABSTRACT-SYNTAX.&Type
      };
}BACnetLogDatum, *PBACnetLogDatum;

*)
	choice	: E_BACnet_LogRecordChoice;
	nRes	: WORD; (* ENUM alignment to 4 byte *)
	aData	: ARRAY[0..4] OF DWORD; (* 20 byte min. size - data type depending on choice selection *)
END_STRUCT
END_TYPE

// DUTs/Types/Properties/[ADS]/LogRecord/ST_BACnet_LogDatumList
{attribute 'hide'}
TYPE ST_BACnet_LogDatumList :
STRUCT
(*

typedef struct _BACnetLogDatumList
{
      DWORD nEntrySize; // 0x80000000 -> next entry
      DWORD reserved;
      BACnetLogDatum listEntry;
}BACnetLogDatumList, *PBACnetLogDatumList;

*)
	nEntrySize	: DWORD; (* 0x80000000 -> next entry *)
	reserved	: DWORD;
	listEntry	: ST_BACnet_LogDatum; (* first entry of log datum list *)
END_STRUCT
END_TYPE

// DUTs/Types/Properties/[ADS]/LogRecord/ST_BACnet_LogRecord
{attribute 'hide'}
TYPE ST_BACnet_LogRecord :
STRUCT
(*

typedef STRUCT _BACnetLogRecord
{
      ULONG validFields;
      BACnetDateTime timestamp;          // [0]
      DWORD statusFlags;                       // [2] optional
      BACnetLogDatumList logDatum;  // [1]
}BACnetLogRecord, *PBACnetLogRecord;

*)
	validFields	: UDINT;
	timestamp	: ST_BA_DateTime;
	statusFlags	: DWORD;
	logDatum	: ST_BACnet_LogDatumList;
END_STRUCT
END_TYPE

// DUTs/Types/Properties/[ADS]/LogRecord/ST_BACnet_LogRecordList
{attribute 'hide'}
TYPE ST_BACnet_LogRecordList :
STRUCT
(*

typedef struct _BACnetLogRecordList
{
      DWORD nEntrySize; // 0x80000000 -> next entry
      DWORD nSequence;  // "reserved"     -> Number of Sequence begins with 1
      BACnetLogRecord listEntry;
}BACnetLogRecordList, *PBACnetLogRecordList;

*)
	nEntrySize	: DWORD; (* 16#80000000 -> next entry *)
	nSequence	: DWORD; (* "reserved"  -> Number OF Sequence begins with 1 *)
	listEntry	: ST_BACnet_LogRecord; (* first entry of record list *)
END_STRUCT
END_TYPE

// DUTs/Types/Properties/[ADS]/Schedule/ST_BACnet_DailySchedule
{attribute 'hide'}
TYPE ST_BACnet_DailySchedule :
STRUCT
(*
	PropWeeklySchedule:
	
	typedef struct _BACnetDailySchedule
	{
	      DWORD nEntrySize; // 0x80000000 -> next entry
	      DWORD reserved;
	      BACnetTimeValueList listEntry;
	} BACnetDailySchedule, *PBACnetDailySchedule;
*)
	nEntrySize	: DWORD;
	nRes		: DWORD;
	stListEntry	: ST_BACnet_TimeValueList;
END_STRUCT
END_TYPE

// DUTs/Types/Properties/[ADS]/Schedule/ST_BACnet_ExceptionScheduleBool
{attribute 'hide'}
TYPE ST_BACnet_ExceptionScheduleBool :
STRUCT
	bReqGet		: BOOL; (* set TRUE if property should reloaded, TRUE --> FALSE = request accepted (starting reload) *)
	bReqSet		: BOOL; (* set TRUE for property write request, TRUE --> FALSE = request accepted (starting storage) *)
	nGet		: USINT; (* reload counter, count up if property was loaded successful *)
	nSet		: USINT; (* save counter, count up if property was stored successful *)
	bBusy		: BOOL; (* started writing data into "arrEntries", don't write data to avoid concurrent access *)
	arrEntries	: ARRAY[0..BACnet_Globals.nDataField_MaxExSchEntries] OF ST_BACnet_ExceptionScheduleEntryBool;
END_STRUCT
END_TYPE

// DUTs/Types/Properties/[ADS]/Schedule/ST_BACnet_ExceptionScheduleCalDate
{attribute 'hide'}
TYPE ST_BACnet_ExceptionScheduleCalDate :
STRUCT
	stStart			: ST_BA_Date;
	stEnd			: ST_BA_Date;
END_STRUCT
END_TYPE

// DUTs/Types/Properties/[ADS]/Schedule/ST_BACnet_ExceptionScheduleCalRef
{attribute 'hide'}
TYPE ST_BACnet_ExceptionScheduleCalRef :
STRUCT
	tCalObjectId	: T_BACnet_ObjectIdentifier := 16#FFFFFFFF;
END_STRUCT
END_TYPE

// DUTs/Types/Properties/[ADS]/Schedule/ST_BACnet_ExceptionScheduleCalWnD
{attribute 'hide'}
TYPE ST_BACnet_ExceptionScheduleCalWnD :
STRUCT
	nMonth			: USINT; (* 255 = all months of year *)
	nWeekOfMonth	: USINT; (* 255 = all weeks of month *)
	nDay			: USINT; (* 255 = all days of month *)
END_STRUCT
END_TYPE

// DUTs/Types/Properties/[ADS]/Schedule/ST_BACnet_ExceptionScheduleEntryBool
{attribute 'hide'}
TYPE ST_BACnet_ExceptionScheduleEntryBool :
STRUCT
	eEntryType		: E_BACnet_CalendarEntryType;
	ePriority		: E_BACnet_Priority;
	stDate			: ST_BACnet_ExceptionScheduleCalDate; (* date / date range *)
	stWeekNDay		: ST_BACnet_ExceptionScheduleCalWnD; (* week and day *)
	stCalRef		: ST_BACnet_ExceptionScheduleCalRef; (* week and day *)
	arrTimeValue	: ARRAY[0..BACnet_Globals.nDataField_MaxTimeValues] OF ST_BACnet_TimeValueBool;
END_STRUCT
END_TYPE

// DUTs/Types/Properties/[ADS]/Schedule/ST_BACnet_ExceptionScheduleEntryReal
{attribute 'hide'}
TYPE ST_BACnet_ExceptionScheduleEntryReal :
STRUCT
	eEntryType		: E_BACnet_CalendarEntryType;
	ePriority		: E_BACnet_Priority;
	stDate			: ST_BACnet_ExceptionScheduleCalDate; (* date / date range *)
	stWeekNDay		: ST_BACnet_ExceptionScheduleCalWnD; (* week and day *)
	stCalRef		: ST_BACnet_ExceptionScheduleCalRef; (* week and day *)
	arrTimeValue	: ARRAY[0..BACnet_Globals.nDataField_MaxTimeValues] OF ST_BACnet_TimeValueReal;
END_STRUCT
END_TYPE

// DUTs/Types/Properties/[ADS]/Schedule/ST_BACnet_ExceptionScheduleReal
{attribute 'hide'}
TYPE ST_BACnet_ExceptionScheduleReal :
STRUCT
	bReqGet		: BOOL; (* set TRUE if property should reloaded, TRUE --> FALSE = request accepted (starting reload) *)
	bReqSet		: BOOL; (* set TRUE for property write request, TRUE --> FALSE = request accepted (starting storage) *)
	nGet		: USINT; (* reload counter, count up if property was loaded successful *)
	nSet		: USINT; (* save counter, count up if property was stored successful *)
	bBusy		: BOOL; (* started writing data into "arrEntries", don't write data to avoid concurrent access *)
	arrEntries	: ARRAY[0..BACnet_Globals.nDataField_MaxExSchEntries] OF ST_BACnet_ExceptionScheduleEntryReal;
END_STRUCT
END_TYPE

// DUTs/Types/Properties/[ADS]/Schedule/ST_BACnet_Value
{attribute 'hide'}
TYPE ST_BACnet_Value :
STRUCT
	eValueChoice	: E_BACnet_ValueChoice;
	nRes1			: WORD; (* ENUM alignment *)
	nSize			: DWORD;
	stValue			: ST_BACnet_EnumerationValueType;
END_STRUCT
END_TYPE

// DUTs/Types/Properties/[ADS]/Schedule/ST_BACnet_ValueList
{attribute 'hide'}
TYPE ST_BACnet_ValueList :
STRUCT
	nEntrySize	: DWORD; (* 0x80000000 -> next entry *)
	reserved	: DWORD;
	listEntry	: ST_BACnet_Value; (* first entry of value list *)
END_STRUCT
END_TYPE

// DUTs/Types/Properties/[ADS]/ST_BACnet_CharacterStringExt
{attribute 'hide'}
TYPE ST_BACnet_CharacterStringExt :
STRUCT
	cookie		: BYTE; (* 0 -> DO differentiate normal strings *)
	encoding	: BYTE;
	strLen		: UINT;
	aData		: ARRAY[1..BACnet_Globals.nBACnetString_MaxLength] OF BYTE;
END_STRUCT
END_TYPE

// DUTs/Types/Properties/[ADS]/ST_BACnet_CharacterStringExtListEntry
{attribute 'hide'}
TYPE ST_BACnet_CharacterStringExtListEntry :
STRUCT
(* list header *)
	nEntrySize	: DWORD; (* byte size of data *)
	hdrInfo		: DWORD;
(* data *)
	extString	: ST_BACnet_CharacterStringExt;
END_STRUCT
END_TYPE

// DUTs/Types/Properties/[ADS]/ST_BACnet_LimitEnable
{attribute 'hide'}
TYPE ST_BACnet_LimitEnable:
STRUCT
	lowLimitEnable : BOOL;
	highLimitEnable : BOOL;
END_STRUCT
END_TYPE

// DUTs/Types/Properties/[ADS]/ST_BACnet_ObjectIdentifierList
{attribute 'hide'}
TYPE ST_BACnet_ObjectIdentifierList :
STRUCT
	nEntries	: UDINT;
	aObjList	: ARRAY[0..BACnet_Globals.nDataField_MaxObjIdList] OF T_BACnet_ObjectIdentifier :=[ 16#FFFFFFFF];
END_STRUCT
END_TYPE

// DUTs/Types/Properties/[Raw]/References/ST_BACnetRaw_DeviceObjectPropertyReference
{attribute 'hide'}
TYPE ST_BACnetRaw_DeviceObjectPropertyReference EXTENDS ST_BACnetRaw_ObjectPropertyReference:
STRUCT
	tDeviceId				: T_BACnet_ObjectIdentifier;
END_STRUCT
END_TYPE

// DUTs/Types/Properties/[Raw]/References/ST_BACnetRaw_DeviceObjectReference
{attribute 'hide'}
TYPE ST_BACnetRaw_DeviceObjectReference :
STRUCT
	nValidFields		: UDINT := 2;
	tDeviceId			: T_BACnet_ObjectIdentifier;
	tObjId				: T_BACnet_ObjectIdentifier;
END_STRUCT
END_TYPE

// DUTs/Types/Properties/[Raw]/References/ST_BACnetRaw_ObjectPropertyReference
{attribute 'hide'}
TYPE ST_BACnetRaw_ObjectPropertyReference :
STRUCT
	stValidFields			: ST_BACnetRaw_ValidFields_DeviceObjectPropertyReference;
	tObjId					: T_BACnet_ObjectIdentifier;
	ePropIdentifier			: E_BACnetPropIdentifier;
	{attribute 'hide'}
	nReserve				: UINT;
	nPropertyArrayIndex		: DWORD;
END_STRUCT
END_TYPE

// DUTs/Types/Properties/[Raw]/References/ST_BACnetRaw_SetpointReference
{attribute 'hide'}
TYPE ST_BACnetRaw_SetpointReference :
STRUCT
	nValidFields	: UDINT;
	stReference		: ST_BACnetRaw_ObjectPropertyReference;
END_STRUCT
END_TYPE

// DUTs/Types/Properties/[Raw]/ValidFields/ST_BACnetRaw_ValidFields_DeviceObjectPropertyReference
{attribute 'hide'}
TYPE ST_BACnetRaw_ValidFields_DeviceObjectPropertyReference :
STRUCT
	bObjectId				: BIT;
	bPropertyIdentifier		: BIT;

	{attribute 'hide'}
	nReserve1				: BIT;
	{attribute 'hide'}
	nReserve2				: BIT;
	{attribute 'hide'}
	nReserve3				: BIT;
	{attribute 'hide'}
	nReserve4				: BIT;
	{attribute 'hide'}
	nReserve5				: BIT;
	{attribute 'hide'}
	nReserve6				: BIT;
	{attribute 'hide'}
	nReserve7				: BYTE;
	{attribute 'hide'}
	nReserve8				: BYTE;
	{attribute 'hide'}
	nReserve9				: BYTE;
END_STRUCT
END_TYPE

// DUTs/Types/Properties/Accumulator/ST_BACnet_Prescale
TYPE ST_BACnet_Prescale :
STRUCT
	nMultiplier		: UDINT		:= 1;
	nModuloDivide	: UDINT		:= 1;
END_STRUCT
END_TYPE

// DUTs/Types/Properties/Accumulator/ST_BACnet_Scale
TYPE ST_BACnet_Scale :
STRUCT
	eChoice		: E_BACnet_ScaleChoice		:= E_BACnet_ScaleChoice.eIntegerScale;
	stValue		: ST_BACnet_ScaleValue		:= (nIntegerScale := 1);
END_STRUCT
END_TYPE

// DUTs/Types/Properties/Accumulator/ST_BACnet_ScaleValue
TYPE ST_BACnet_ScaleValue :
UNION
	fFloatScale		: REAL;
	nIntegerScale	: DINT;	
END_UNION
END_TYPE

// DUTs/Types/Properties/Calendar/T_BACnet_CalendarDateList
TYPE T_BACnet_CalendarDateList : ARRAY[1 .. BACnet_Param.nCal_DateListCount] OF ST_BA_CalendarEntry; END_TYPE

// DUTs/Types/Properties/Event/ST_BACnet_Event
TYPE ST_BACnet_Event :
STRUCT
	bAcked			: BOOL;
	sMessage		: STRING;
	dtTimeStamp		: DT;
	
	{attribute 'hide'} 
    {attribute 'tc_no_symbol'}
	stBACnetTime	: ST_BACnet_TimeStampDateTime;
END_STRUCT
END_TYPE

// DUTs/Types/Properties/Event/ST_BACnet_EventMessageTexts
TYPE ST_BACnet_EventMessageTexts :
STRUCT
	stToOffNormal	: ST_BACnet_CharacterStringExtListEntry;
	stToFault		: ST_BACnet_CharacterStringExtListEntry;
	stToNormal		: ST_BACnet_CharacterStringExtListEntry;
END_STRUCT
END_TYPE

// DUTs/Types/Properties/Event/ST_BACnet_EventMessageTextStrings
TYPE ST_BACnet_EventMessageTextStrings :
STRUCT
	sToOffNormal	: STRING;
	sToFault		: STRING;
	sToNormal		: STRING;
END_STRUCT
END_TYPE

// DUTs/Types/Properties/Event/ST_BACnet_Events
TYPE ST_BACnet_Events :
STRUCT
	stToOffNormal	: ST_BACnet_Event;
	stToFault		: ST_BACnet_Event;
	stToNormal		: ST_BACnet_Event;
END_STRUCT
END_TYPE

// DUTs/Types/Properties/Event/ST_BACnet_EventTimeStamps
TYPE ST_BACnet_EventTimeStamps :
STRUCT
	stToOffNormal	: ST_BACnet_TimeStampDateTime;
	stToFault		: ST_BACnet_TimeStampDateTime;
	stToNormal		: ST_BACnet_TimeStampDateTime;
END_STRUCT
END_TYPE

// DUTs/Types/Properties/Event/T_BACnet_EventTransitions
TYPE T_BACnet_EventTransitions : ARRAY[E_BA_EventTransition.First .. E_BA_EventTransition.Last] OF BOOL; END_TYPE

// DUTs/Types/Properties/Event/T_BACnet_EventTransitionTexts
TYPE T_BACnet_EventTransitionTexts : ARRAY[E_BA_EventTransition.First .. E_BA_EventTransition.Last] OF T_MaxString; END_TYPE

// DUTs/Types/Properties/EventEnrollment/ST_BACnet_EventArguments
TYPE ST_BACnet_EventArguments :
UNION
	stOutOfRange		: ST_BACnet_EventOutOfRange;
	stUnsignedRange		: ST_BACnet_EventUnsignedRange;
	stBinaryCoded		: ST_BACnet_EventBinaryCoded;
END_UNION
END_TYPE

// DUTs/Types/Properties/EventEnrollment/ST_BACnet_EventBinaryCoded
TYPE ST_BACnet_EventBinaryCoded :
STRUCT
	aData : ARRAY [0..BACnet_Param.nEE_EventParameter_BinaryCodedSize] OF BYTE;
END_STRUCT
END_TYPE

// DUTs/Types/Properties/EventEnrollment/ST_BACnet_EventOutOfRange
TYPE ST_BACnet_EventOutOfRange :
STRUCT
	nTimeDelay : UDINT;
	fLowLimit  : REAL;
	fHighLimit : REAL;
	fDeadband  : REAL;
END_STRUCT
END_TYPE

// DUTs/Types/Properties/EventEnrollment/ST_BACnet_EventParameter
TYPE ST_BACnet_EventParameter :
STRUCT
	eEventType		: E_BACnet_EventType;
	{attribute 'hide'} 
    {attribute 'tc_no_symbol'}
	nReserved1		: INT;
	nArgSize 		: DINT;							// reserved in stack, used for saving size in plc
	stEventArgs		: ST_BACnet_EventArguments;
END_STRUCT
END_TYPE

// DUTs/Types/Properties/EventEnrollment/ST_BACnet_EventUnsignedRange
TYPE ST_BACnet_EventUnsignedRange :
STRUCT
	{attribute 'parameterUnit':= 's'}
	nTimedelay		: UDINT;				// in [s]
	nLowLimit		: UDINT;
	nHighLimit		: UDINT;
END_STRUCT
END_TYPE

// DUTs/Types/Properties/Recipient/ST_BACnet_Address
{attribute 'hide'}
TYPE ST_BACnet_Address :
STRUCT
	eChoice		: E_BACnet_AddressChoice;
	{attribute 'hide'}
	nReserve1	: UINT;
	aAddress	: ARRAY [0..7] OF BYTE;
	nNetworkNr	: UINT;
END_STRUCT
END_TYPE

// DUTs/Types/Properties/Recipient/ST_BACnet_Destination
{attribute 'hide'}
TYPE ST_BACnet_Destination :
STRUCT
	stValidDays			: ST_BACnet_ValidDays;
	{attribute 'hide'}
	nReserve1			: UINT; 
	stFromTime			: ST_BA_Time						:= F_BA_ToSTTime(T#0H);
	stToTime			: ST_BA_Time						:= F_BA_ToSTTime(T#23H59M59S);
	stRecipient			: ST_BACnet_Recipient;
	nProcessId			: UDINT;
	nEventTransitions	: ST_BACnet_EventTransitionBits;
	{attribute 'hide'}
	nReserve2			: UINT; 
	bIssueConfirmed		: BOOL;
	{attribute 'hide'}
	nReserve3			: ARRAY[0..2] OF BYTE;
END_STRUCT
END_TYPE

// DUTs/Types/Properties/Recipient/ST_BACnet_Recipient
{attribute 'hide'}
TYPE ST_BACnet_Recipient :
STRUCT
	eRecipientChoice	: E_BACnet_RecipientChoice;
	{attribute 'hide'}
	nReserve1			: UINT := 0;
	stEntry 			: ST_BACnet_RecipientEntry;
END_STRUCT
END_TYPE

// DUTs/Types/Properties/Recipient/ST_BACnet_RecipientEntry
{attribute 'hide'}
TYPE ST_BACnet_RecipientEntry :
UNION
	nDeviceInstance		: UDINT;
//	tDeviceId			: T_BACnet_ObjectIdentifier := 16#FFFFFFFF;
	stNetAddr			: ST_BACnet_Address;
END_UNION
END_TYPE

// DUTs/Types/Properties/Recipient/ST_BACnet_ValidDays
{attribute 'hide'}
TYPE ST_BACnet_ValidDays :
STRUCT
	{attribute 'hide'}
	nReserve1		: BYTE;	
	{attribute 'hide'}
	nReserve2		: BIT;
	
	bSunday			: BIT;
	bSaturday		: BIT;
	bFriday			: BIT;
	bThursday		: BIT;
	bWednesday		: BIT;
	bTuesday		: BIT;
	bMonday			: BIT;
END_STRUCT
END_TYPE

// DUTs/Types/Properties/Recipient/T_BACnet_RecipientList
TYPE T_BACnet_RecipientList : ARRAY [1 .. BACnet_Param.nNC_RecipientListSize] OF ST_BACnet_Destination; END_TYPE

// DUTs/Types/Properties/References/ST_BACnet_ObjectPropertyReference
TYPE ST_BACnet_ObjectPropertyReference :
STRUCT
	iObject				: I_BACnet_Object;
	tObjectID			: T_BACnet_ObjectIdentifier		:= 16#FFFFFFFF;
	ePropertyId			: E_BACnetPropIdentifier		:= E_BACnetPropIdentifier.PropPresentValue;
END_STRUCT
END_TYPE

// DUTs/Types/Properties/Scheduler/ST_BACnet_EnumerationValueType
TYPE ST_BACnet_EnumerationValueType :
STRUCT
	eChoice			: E_BACnet_EnumerationValueChoice;
	nEnumValue		: UDINT;
END_STRUCT
END_TYPE

// DUTs/Types/Properties/Scheduler/ST_BACnet_SchedCalendar
TYPE ST_BACnet_SchedCalendar :
STRUCT
	iRefCalendar	: I_BACnet_Object;
	tRefCalendarID	: T_BACnet_ObjectIdentifier := BACnet_Globals.nBACnetObjId_None;
	
	{attribute 'hide'}
	nReserve1		: DWORD; // May be used in future as a sequence-index
	
	eEventPriority	: E_BACnet_Priority := E_BACnet_Priority.eP1;
	aEntry			: ARRAY[1 .. BACnet_Param.nSched_EntryCount] OF ST_BA_SchedEntry;
END_STRUCT
END_TYPE

// DUTs/Types/Properties/Scheduler/ST_BACnet_SchedException
TYPE ST_BACnet_SchedException :
STRUCT
	eType			: E_BA_DateValChoice := E_BA_DateValChoice.Invalid;
	uDate			: U_BA_DateVal;
	
	{attribute 'hide'}
	nReserve		: DWORD;			// May be used in future as a sequence-index
	
	nEventPriority	: UDINT := 1;
	aEntry			: T_BACnet_SchedExceptionEntryList;
END_STRUCT
END_TYPE

// DUTs/Types/Properties/Scheduler/ST_BACnet_SpecialEvent
TYPE ST_BACnet_SpecialEvent :
STRUCT
	eEventChoice		: E_BACnet_SpecialEventChoice;
	{attribute 'hide'}
	nReserve1			: UINT;
	eCalEntryChoice		: E_BACnet_CalendarEntryChoice;
	{attribute 'hide'}
	nReserve2			: UINT;
	uCalEntry			: U_BA_DateVal;				// BACnetObjectIdentifier calendarReference;
	nEventPriority		: UDINT;
	{attribute 'hide'}
	nReserve3			: UDINT;
END_STRUCT
END_TYPE

// DUTs/Types/Properties/Scheduler/ST_BACnet_SpecialEventList
TYPE ST_BACnet_SpecialEventList :
STRUCT
	nEntrySize	: DWORD;
	nRes		: DWORD;
	stEvent 	: ST_BACnet_SpecialEvent;
END_STRUCT
END_TYPE

// DUTs/Types/Properties/Scheduler/T_BACnet_SchedCalendar
TYPE T_BACnet_SchedCalendar : ARRAY[1 .. BACnet_Param.nSched_CalendarCount] OF ST_BACnet_SchedCalendar; END_TYPE

// DUTs/Types/Properties/Scheduler/T_BACnet_SchedExceptionEntryList
TYPE T_BACnet_SchedExceptionEntryList : ARRAY[1 .. BACnet_Param.nSched_EntryCount] OF ST_BA_SchedEntry; END_TYPE

// DUTs/Types/Properties/Scheduler/T_BACnet_SchedExceptionList
TYPE T_BACnet_SchedExceptionList : ARRAY[1 .. BACnet_Param.nSched_ExceptionCount] OF ST_BACnet_SchedException; END_TYPE

// DUTs/Types/Properties/Scheduler/T_BACnet_SchedWeek
TYPE T_BACnet_SchedWeek : ARRAY[E_BA_Weekday.First .. E_BA_Weekday.Last, 1 .. BACnet_Param.nSched_EntryCount] OF ST_BA_SchedEntry; END_TYPE

// DUTs/Types/Properties/TLog/T_BACnet_TLogBuffer
TYPE T_BACnet_TLogBuffer : ARRAY [1 .. BACnet_Param.nLog_BufferEntryCount] OF ST_BA_TrendEntry; END_TYPE

// DUTs/Types/Properties/ST_BACnet_ClientCOV
TYPE ST_BACnet_ClientCOV :
STRUCT
	eChoice : E_BACnet_ClientCOVChoice := E_BACnet_ClientCOVChoice.eCovNull;
	{attribute 'hide'}
	nReserved		: UINT;
	fIncrement		: REAL;
END_STRUCT
END_TYPE

// DUTs/Types/Properties/ST_BACnet_EventTransitionBits
{attribute 'hide'}
TYPE ST_BACnet_EventTransitionBits :
STRUCT
	{attribute 'hide'}
	_nUnusedBits	: BYTE := 5;
	
	{attribute 'hide'}
	nReserve1		: BIT;
	{attribute 'hide'}
	nReserve2		: BIT;
	{attribute 'hide'}
	nReserve3		: BIT;
	{attribute 'hide'}
	nReserve4		: BIT;
	{attribute 'hide'}
	nReserve5		: BIT;
	
	bToNormal		: BIT;
	bToFault		: BIT;
	bToOffNormal	: BIT;
END_STRUCT
END_TYPE

// DUTs/Types/Properties/ST_BACnet_LimitEnableBits
{attribute 'hide'}
TYPE ST_BACnet_LimitEnableBits :
STRUCT
	{attribute 'hide'}
	_nUnusedBits		: BYTE := 6;
	
	{attribute 'hide'}
	nReserve1			: BIT;
	{attribute 'hide'}
	nReserve2			: BIT;
	{attribute 'hide'}
	nReserve3			: BIT;
	{attribute 'hide'}
	nReserve4			: BIT;
	{attribute 'hide'}
	nReserve5			: BIT;
	{attribute 'hide'}
	nReserve6			: BIT;
	
	bHighLimitEnable	: BIT;
	bLowLimitEnable		: BIT;
END_STRUCT
END_TYPE

// DUTs/Types/Properties/ST_BACnet_ServicesSupportedBits
{attribute 'hide'}
TYPE ST_BACnet_ServicesSupportedBits :
STRUCT
	{attribute 'hide'}
	nReserve1			: BYTE;
	
	bSuppAtomicWriteFile  : BIT;
	bSuppAtomicReadFile  : BIT;
	bSuppSubscribeCOV  : BIT;
	bSuppGetEnrollmentSummary  : BIT;
	bSuppGetAlarmSummary  : BIT;
	bSuppConfirmedEventNotification  : BIT;
	bSuppConfirmedCOVNotification  : BIT;	
	bSuppAcknowledgeAlarm : BIT;

	bSuppWriteProperty : BIT;
	bSuppReadPropertyMultiple  : BIT;
	bSuppReadPropertyConditional  : BIT;
	bSuppReadProperty  : BIT;
	bSuppDeleteObject : BIT;
	bSuppCreateObject  : BIT;
	bSuppRemoveListElement  : BIT;
	bSuppAddListElement  : BIT;

	bSuppVtData  : BIT;
	bSuppVtClose : BIT;
	bSuppVtOpen  : BIT;
	bSuppReinitializeDevice  : BIT;	
	bSuppConfirmedTextMessage : BIT;
	bSuppConfirmedPrivateTransfer : BIT;
	bSuppDeviceCommunicationControl  : BIT;
	bSuppWritePropertyMultiple  : BIT;

	bSuppUnconfirmedTextMessage  : BIT;
	bSuppUnconfirmedPrivateTransfer  : BIT;
	bSuppUnconfirmedEventNotification  : BIT;	
	bSuppUnconfirmedCOVNotification  : BIT;
	bSuppIHave  : BIT;
	bSuppIAm  : BIT;
	bSuppRequestKey  : BIT;	
	bSuppAuthenticate  : BIT;

	bSuppGetEventInformation  : BIT;
	bSuppSubscribeCOVProperty  : BIT;
	bSuppLifeSafetyOperation  : BIT;
	bSuppUtcTimeSynchronization  : BIT;
	bSuppReadRange  : BIT;
	bSuppWhoIs  : BIT;
	bSuppWhoHas  : BIT;	
	bSuppTimeSynchronization  : BIT;
	
	{attribute 'hide'}
	nReserve2			: BYTE;
END_STRUCT
END_TYPE

// DUTs/Types/Properties/ST_BACnet_StatusFlagBits
TYPE ST_BACnet_StatusFlagBits :
STRUCT
	{attribute 'hide'}
	_nUnusedBits	: BYTE;
	
	{attribute 'hide'}
	nReserve1		: BIT;
	{attribute 'hide'}
	nReserve2		: BIT;
	{attribute 'hide'}
	nReserve3		: BIT;
	{attribute 'hide'}
	nReserve4		: BIT;
	
	bAlarm			: BIT;
	bFault			: BIT;
	bOverriden		: BIT;
	bOutOfSerice	: BIT;
END_STRUCT
END_TYPE

// DUTs/Types/Properties/T_BACnet_EventTransitionPriority
TYPE T_BACnet_EventTransitionPriority : ARRAY[E_BA_EventTransition.First .. E_BA_EventTransition.Last] OF UDINT(0 .. 255); END_TYPE

// DUTs/Types/Properties/T_BACnet_ObjectIdentifier
TYPE T_BACnet_ObjectIdentifier : DWORD; END_TYPE

// DUTs/Types/Properties/T_BACnet_StateText
TYPE T_BACnet_StateText : STRING(BACnet_Param.nStateText_Length); END_TYPE

// DUTs/Types/Properties/T_BACnet_StateTextArray
TYPE T_BACnet_StateTextArray : ARRAY[1 .. BACnet_Param.nMultistate_StateCount] OF T_BACnet_StateText; END_TYPE

// DUTs/Types/Remote/[Internal]/ST_BACnetRM_CmdRealValue
{attribute 'hide'} // [Workaround] Not hidden when lib is included

TYPE INTERNAL ST_BACnetRM_CmdRealValue :
STRUCT
	fValue : REAL;
	bNull : BOOL;
END_STRUCT
END_TYPE

// DUTs/Types/Remote/[Internal]/ST_BACnetRM_FifoEntry
{attribute 'hide'} // [Workaround] Not hidden when lib is included

TYPE INTERNAL ST_BACnetRM_FifoEntry :
UNION
	fbRead : POINTER TO FB_BACnetRM_ReadProperty;
	fbWrite : POINTER TO FB_BACnetRM_WriteProperty;
END_UNION
END_TYPE

// DUTs/Types/Remote/[Internal]/ST_BACnetRM_LastWriteValue
{attribute 'hide'} // [Workaround] Not hidden when lib is included

TYPE INTERNAL ST_BACnetRM_LastWriteValue :
UNION
	stCmdValue : ST_BACnetRM_CmdRealValue;
	n8Value : BYTE;
	n16Value : UINT;
	n32Value : UDINT;
	nOther : POINTER TO BYTE;
END_UNION
END_TYPE

// DUTs/Types/Remote/[Internal]/ST_BACnetRM_PropertyValueList
{attribute 'hide'} // [Workaround] Not hidden when lib is included

{attribute 'enable_dynamic_creation'}
TYPE INTERNAL ST_BACnetRM_PropertyValueList :
STRUCT
	nEntrySize		: DWORD; (* 0x80000000 -> next entry *)
	{attribute 'hide'}
	nRes			: DWORD;
	nValidFields	: DWORD;
	ePropID			: E_BACnetPropIdentifier;		// [0]
	nArrayIndex		: DWORD;						// [1] (Optional)
	nPriority		: DWORD;						// [3] Unsigned (1 .. 16) (Optional -- used only when property is commandable)
	nValueSize		: DWORD;
	nDataType		: DWORD;
	
	// Data
END_STRUCT
END_TYPE

// DUTs/Types/Remote/[Internal]/ST_BACnetRM_ReadEntry
{attribute 'hide'} // [Workaround] Not hidden when lib is included

{attribute 'enable_dynamic_creation'}
TYPE INTERNAL ST_BACnetRM_ReadEntry :
STRUCT
	iObject 		: I_BACnetRM_BaseObject;
	ePropID 		: E_BACnetPropIdentifier;
	
	nData 			: UDINT;
	pData 			: PVOID;
	nIndex 			: UDINT := 16#FFFFFFFF;
	
	iReadFB 		: I_BACnetRM_BasicReq;
	
	_bError			: BOOL;										// Temporary error flag
	
